# B&R Automation Studio project Panasonic_LinkaPowerCP2_A2021055 (part 31)

#### COM_Tester.st
```iecst
ACTION COM_Tester:

	//Parametre komunikácie//
    memcpy(ADR(SKTcpClientTester_0.Params.IPaddrServ),ADR('192.168.128.252'),SIZEOF('192.168.128.252'));
    (*memcpy(ADR(SKTcpClientTester_0.Params.IPaddrServ),ADR('127.0.0.1'),SIZEOF('127.0.0.1'));*)
    SKTcpClientTester_0.Params.IPportClient := P4_FunkcnyTestA.PAR.CisloPortuKlienta;
    SKTcpClientTester_0.Params.IPportServ := 1030;
    SKTcpClientTester_0.Params.RecvTimeout := 10000;
    strcpy(ADR(SKTcpClientTester_0.Params.Packet.data),ADR(dataStr));
    SKTcpClientTester_0();

    Cas_FunkcnyTestA.PT:= T#1M;
    Cas_FunkcnyTestA();

    //Volanie funkcie SequenceControl//
    SequenceControl(SC:= SC_OvlTesteraFT);

    CASE SC_OvlTesteraFT.Step OF

        0:
            SC_OvlTesteraFT.StepName:= '0 - Nulovanie';
            SKTcpClientTester_0.Enable:= TRUE;
            SKTcpClientTester_0.Cmd.Send:= FALSE;
			P4_FunkcnyTestA.STAV.TestovanieUkoncene:= FALSE;
			P4_FunkcnyTestA.STAV.TesterNeodpoveda:= FALSE;
            PocetDopytovNaTester:= 0;
            SC_OvlTesteraFT.ResetStep:= TRUE;
            SC_OvlTesteraFT.Step:= 1;

        1:
            SC_OvlTesteraFT.StepName:= '1 - Cakam na spustenie testera';
            IF P4_FunkcnyTestA.CMD.StartTestovania THEN
                P4_FunkcnyTestA.STAV.Vysledok_FV_Testu:= '';
                Cas_FunkcnyTestA.IN:= TRUE;
                NameranyCasFunkcnehoTestuA:= 0;
                SC_OvlTesteraFT.Step:= 10;
            END_IF

        10:
            SC_OvlTesteraFT.StepName:= '10 - Dopyt na stav testera - typ 0';
            SC_OvlTesteraFT.IdleTime.PT:= T#300ms;
            SC_OvlTesteraFT.AlarmTime.PT:= T#5s;
            SC_OvlTesteraFT.IdleTime.IN:= TRUE;
            SC_OvlTesteraFT.AlarmTime.IN:= TRUE;

            SKTcpClientTester_0.Params.Packet.type:= 0;
            SKTcpClientTester_0.Params.Packet.workplace:= 49;
            SKTcpClientTester_0.Params.Packet.id:= 1;
            SKTcpClientTester_0.Cmd.Close:= FALSE;
			SKTcpClientTester_0.Cmd.Send:= TRUE;

            IF SKTcpClientTester_0.Cmd.Send AND NOT SKTcpClientTester_0.Status.staReceived AND NOT SKTcpClientTester_0.Status.staError THEN
                SC_OvlTesteraFT.ResetStep:= TRUE;
                SC_OvlTesteraFT.Step:= 13;
            ELSIF SC_OvlTesteraFT.AlarmTime.Q AND (SKTcpClientTester_0.Status.staReceived OR SKTcpClientTester_0.Status.staError) THEN
                PocetDopytovNaTester:= PocetDopytovNaTester + 1;
				SKTcpClientTester_0.Cmd.Send:= FALSE;
				SKTcpClientTester_0.Cmd.Close:= TRUE;
				SC_OvlTesteraFT.ResetStep:= TRUE;
                SC_OvlTesteraFT.Step:= 12;
            END_IF

        12:
            SC_OvlTesteraFT.StepName:= '12 - Dopyt na stav testera - cakam na opatovny dopyt na tester';
            SC_OvlTesteraFT.IdleTime.PT:= T#800ms;
            SC_OvlTesteraFT.AlarmTime.PT:= T#5s;
            SC_OvlTesteraFT.IdleTime.IN:= TRUE;
            SKTcpClientTester_0.Cmd.Send:= FALSE;

            IF PocetDopytovNaTester < 10 THEN
                IF SC_OvlTesteraFT.IdleTime.Q THEN
                    SC_OvlTesteraFT.ResetStep:= TRUE;
                    SC_OvlTesteraFT.Step:= 10;
                END_IF
            ELSE
                P4_FunkcnyTestA.STAV.Vysledok_FV_Testu:= 'NG';
                P4_FunkcnyTestA.STAV.TesterNeodpoveda:= TRUE;
                SC_OvlTesteraFT.ResetStep:= TRUE;
                SC_OvlTesteraFT.Step:= 100;
            END_IF

        13:
            SC_OvlTesteraFT.StepName:= '13 - Odpoved na stav testera - typ 0';
            SC_OvlTesteraFT.IdleTime.PT:= T#800ms;
            SC_OvlTesteraFT.AlarmTime.PT:= T#10s;
            SC_OvlTesteraFT.IdleTime.IN:= TRUE;

            IF SKTcpClientTester_0.Status.staReceived AND SKTcpClientTester_0.Status.DataRecv[2]= 0 AND SKTcpClientTester_0.Status.DataRecv[5]= 2 THEN
                SKTcpClientTester_0.Cmd.Send:= FALSE;
                SC_OvlTesteraFT.ResetStep:= TRUE;
                SC_OvlTesteraFT.Step:= 15;
            ELSIF SKTcpClientTester_0.Status.staReceived AND SKTcpClientTester_0.Status.DataRecv[2]= 0 AND SKTcpClientTester_0.Status.DataRecv[5]= 1 THEN
				SKTcpClientTester_0.Cmd.Send:= FALSE;
				SKTcpClientTester_0.Cmd.Close:= TRUE;
                IF SC_OvlTesteraFT.IdleTime.Q THEN
                    SC_OvlTesteraFT.ResetStep:= TRUE;
                    SC_OvlTesteraFT.Step:= 10;
                END_IF
            ELSIF SKTcpClientTester_0.Status.staReceived AND SKTcpClientTester_0.Status.DataRecv[2]= 0 AND SKTcpClientTester_0.Status.DataRecv[5]= 0 THEN
                SKTcpClientTester_0.Cmd.Send:= FALSE;
                SKTcpClientTester_0.Cmd.Close:= TRUE;
				IF SC_OvlTesteraFT.IdleTime.Q THEN
                    SC_OvlTesteraFT.ResetStep:= TRUE;
                    SC_OvlTesteraFT.Step:= 10;
                END_IF
            ELSIF SKTcpClientTester_0.Status.staError THEN
                SKTcpClientTester_0.Cmd.Send:= FALSE;
                P4_FunkcnyTestA.STAV.Vysledok_FV_Testu:= 'NG';
                P4_FunkcnyTestA.STAV.TesterNeodpoveda:= TRUE;
                SC_OvlTesteraFT.ResetStep:= TRUE;
                SC_OvlTesteraFT.Step:= 100;
            END_IF

        15:
            SC_OvlTesteraFT.StepName:= '15 - Poslanie QR kodu Power CP - typ 1';
            SC_OvlTesteraFT.IdleTime.PT:= T#300ms;
            SC_OvlTesteraFT.AlarmTime.PT:= T#10s;
            SC_OvlTesteraFT.IdleTime.IN:= TRUE;

            SKTcpClientTester_0.Params.Packet.type:= 1;
            SKTcpClientTester_0.Params.Packet.workplace:= 49;
            SKTcpClientTester_0.Params.Packet.id:= 1;
			dataStr:= Paletka[i].PAR.QRkodPowerCP;
		    SKTcpClientTester_0.Cmd.Send:= TRUE;

            IF SKTcpClientTester_0.Cmd.Send AND NOT SKTcpClientTester_0.Status.staReceived AND NOT SKTcpClientTester_0.Status.staError THEN
                SC_OvlTesteraFT.ResetStep:= TRUE;
                SC_OvlTesteraFT.Step:= 18;
            END_IF

        18:
            SC_OvlTesteraFT.StepName:= '18 - Odpoved na poslanie QR kodu - typ 1';
            SC_OvlTesteraFT.IdleTime.PT:= T#300ms;
            SC_OvlTesteraFT.AlarmTime.PT:= T#10s;
            SC_OvlTesteraFT.IdleTime.IN:= TRUE;

            IF SKTcpClientTester_0.Status.staReceived AND SKTcpClientTester_0.Status.DataRecv[2]= 1 AND SKTcpClientTester_0.Status.DataRecv[5]= 0 THEN
                SKTcpClientTester_0.Cmd.Send:= FALSE;
                SC_OvlTesteraFT.ResetStep:= TRUE;
                SC_OvlTesteraFT.Step:= 20;
            ELSIF SKTcpClientTester_0.Status.staReceived AND SKTcpClientTester_0.Status.DataRecv[2]= 1 AND SKTcpClientTester_0.Status.DataRecv[5]= 2 THEN
                SKTcpClientTester_0.Cmd.Send:= FALSE;
                IF SC_OvlTesteraFT.IdleTime.Q THEN
                    SC_OvlTesteraFT.ResetStep:= TRUE;
                    SC_OvlTesteraFT.Step:= 15;
                END_IF
            ELSIF SKTcpClientTester_0.Status.staReceived AND SKTcpClientTester_0.Status.DataRecv[2]= 1 AND SKTcpClientTester_0.Status.DataRecv[5]= 1 THEN
                SKTcpClientTester_0.Cmd.Send:= FALSE;
                P4_FunkcnyTestA.STAV.Vysledok_FV_Testu:= 'NG';
                P4_FunkcnyTestA.STAV.TestovanieUkoncene:= TRUE;
                SC_OvlTesteraFT.ResetStep:= TRUE;
                SC_OvlTesteraFT.Step:= 100;
            ELSIF SKTcpClientTester_0.Status.staError THEN
                SKTcpClientTester_0.Cmd.Send:= FALSE;
                P4_FunkcnyTestA.STAV.Vysledok_FV_Testu:= 'NG';
                P4_FunkcnyTestA.STAV.TesterNeodpoveda:= TRUE;
                SC_OvlTesteraFT.ResetStep:= TRUE;
                SC_OvlTesteraFT.Step:= 100;
            END_IF

        20:
            SC_OvlTesteraFT.StepName:= '20 - Dopyt na stav testera - typ 0';
            SC_OvlTesteraFT.IdleTime.PT:= T#300ms;
            SC_OvlTesteraFT.AlarmTime.PT:= T#10s;
            SC_OvlTesteraFT.IdleTime.IN:= TRUE;

            SKTcpClientTester_0.Params.Packet.type:= 0;
            SKTcpClientTester_0.Params.Packet.workplace:= 49;
            SKTcpClientTester_0.Params.Packet.id:= 1;
            SKTcpClientTester_0.Cmd.Send:= TRUE;

            IF SKTcpClientTester_0.Cmd.Send AND NOT SKTcpClientTester_0.Status.staReceived AND NOT SKTcpClientTester_0.Status.staError THEN
                SC_OvlTesteraFT.ResetStep:= TRUE;
                SC_OvlTesteraFT.Step:= 23;
            END_IF

        23:
            SC_OvlTesteraFT.StepName:= '23 - Odpoved na stav testera - typ 0';
            SC_OvlTesteraFT.IdleTime.PT:= T#300ms;
            SC_OvlTesteraFT.AlarmTime.PT:= T#10s;
            SC_OvlTesteraFT.IdleTime.IN:= TRUE;

            IF SKTcpClientTester_0.Status.staReceived AND SKTcpClientTester_0.Status.DataRecv[2]= 0 AND SKTcpClientTester_0.Status.DataRecv[5]= 3 THEN
                SKTcpClientTester_0.Cmd.Send:= FALSE;
                IF SC_OvlTesteraFT.IdleTime.Q THEN
                    SC_OvlTesteraFT.ResetStep:= TRUE;
                    SC_OvlTesteraFT.Step:= 20;
                END_IF
            ELSIF SKTcpClientTester_0.Status.staReceived AND SKTcpClientTester_0.Status.DataRecv[2]= 0 AND SKTcpClientTester_0.Status.DataRecv[5]= 4 THEN
                SKTcpClientTester_0.Cmd.Send:= FALSE;
                SC_OvlTesteraFT.ResetStep:= TRUE;
                SC_OvlTesteraFT.Step:= 25;
            ELSIF SKTcpClientTester_0.Status.staReceived AND SKTcpClientTester_0.Status.DataRecv[2]= 0 AND SKTcpClientTester_0.Status.DataRecv[5]= 0 THEN
                SKTcpClientTester_0.Cmd.Send:= FALSE;
                P4_FunkcnyTestA.STAV.Vysledok_FV_Testu:= 'NG';
                P4_FunkcnyTestA.STAV.TestovanieUkoncene:= TRUE;
                SC_OvlTesteraFT.ResetStep:= TRUE;
                SC_OvlTesteraFT.Step:= 100;
            ELSIF SKTcpClientTester_0.Status.staError THEN
                SKTcpClientTester_0.Cmd.Send:= FALSE;
                P4_FunkcnyTestA.STAV.Vysledok_FV_Testu:= 'NG';
                P4_FunkcnyTestA.STAV.TesterNeodpoveda:= TRUE;
                SC_OvlTesteraFT.ResetStep:= TRUE;
                SC_OvlTesteraFT.Step:= 100;
            END_IF

        25:
            SC_OvlTesteraFT.StepName:= '25 - Dopyt na vysledok testu - typ 2';
            SC_OvlTesteraFT.IdleTime.PT:= T#300ms;
            SC_OvlTesteraFT.AlarmTime.PT:= T#10s;
            SC_OvlTesteraFT.IdleTime.IN:= TRUE;

            SKTcpClientTester_0.Params.Packet.type:= 2;
            SKTcpClientTester_0.Params.Packet.workplace:= 49;
            SKTcpClientTester_0.Params.Packet.id:= 1;
            SKTcpClientTester_0.Cmd.Send:= TRUE;

            IF SKTcpClientTester_0.Cmd.Send AND NOT SKTcpClientTester_0.Status.staReceived AND NOT SKTcpClientTester_0.Status.staError THEN
                SC_OvlTesteraFT.ResetStep:= TRUE;
                SC_OvlTesteraFT.Step:= 28;
            END_IF

        28:
            SC_OvlTesteraFT.StepName:= '28 - Odpoved na vysledok testu - typ 2';
            SC_OvlTesteraFT.IdleTime.PT:= T#300ms;
            SC_OvlTesteraFT.AlarmTime.PT:= T#10s;
            SC_OvlTesteraFT.IdleTime.IN:= TRUE;

            IF SKTcpClientTester_0.Status.staReceived AND SKTcpClientTester_0.Status.DataRecv[2]= 2 AND SKTcpClientTester_0.Status.DataRecv[5]= 1 THEN
                SKTcpClientTester_0.Cmd.Send:= FALSE;
                P4_FunkcnyTestA.STAV.Vysledok_FV_Testu:= 'OK';
                SC_OvlTesteraFT.ResetStep:= TRUE;
                SC_OvlTesteraFT.Step:= 30;
            ELSIF SKTcpClientTester_0.Status.staReceived AND SKTcpClientTester_0.Status.DataRecv[2]= 2 AND SKTcpClientTester_0.Status.DataRecv[5]= 2 THEN
                SKTcpClientTester_0.Cmd.Send:= FALSE;
                P4_FunkcnyTestA.STAV.Vysledok_FV_Testu:= 'NG';
                SC_OvlTesteraFT.ResetStep:= TRUE;
                SC_OvlTesteraFT.Step:= 30;
            ELSIF SKTcpClientTester_0.Status.staReceived AND SKTcpClientTester_0.Status.DataRecv[2]= 2 AND SKTcpClientTester_0.Status.DataRecv[5]= 0 THEN
                SKTcpClientTester_0.Cmd.Send:= FALSE;
                IF SC_OvlTesteraFT.IdleTime.Q THEN
                    SC_OvlTesteraFT.ResetStep:= TRUE;
                    SC_OvlTesteraFT.Step:= 25;
                END_IF
            ELSIF SKTcpClientTester_0.Status.staReceived AND SKTcpClientTester_0.Status.DataRecv[2]= 2 AND SKTcpClientTester_0.Status.DataRecv[5]= 3 THEN
                SKTcpClientTester_0.Cmd.Send:= FALSE;
                IF SC_OvlTesteraFT.IdleTime.Q THEN
                    SC_OvlTesteraFT.ResetStep:= TRUE;
                    SC_OvlTesteraFT.Step:= 25;
                END_IF
            ELSIF SKTcpClientTester_0.Status.staError THEN
                SKTcpClientTester_0.Cmd.Send:= FALSE;
                P4_FunkcnyTestA.STAV.Vysledok_FV_Testu:= 'NG';
                P4_FunkcnyTestA.STAV.TesterNeodpoveda:= TRUE;
                SC_OvlTesteraFT.ResetStep:= TRUE;
                SC_OvlTesteraFT.Step:= 100;
            END_IF

        30:
            SC_OvlTesteraFT.StepName:= '30 - Potvrdenie precitanie vysledkov testu - typ 3';
            SC_OvlTesteraFT.IdleTime.PT:= T#300ms;
            SC_OvlTesteraFT.AlarmTime.PT:= T#10s;
            SC_OvlTesteraFT.IdleTime.IN:= TRUE;

            SKTcpClientTester_0.Params.Packet.type:= 3;
            SKTcpClientTester_0.Params.Packet.workplace:= 49;
            SKTcpClientTester_0.Params.Packet.id:= 1;
            SKTcpClientTester_0.Cmd.Send:= TRUE;

            IF SKTcpClientTester_0.Cmd.Send AND NOT SKTcpClientTester_0.Status.staReceived AND NOT SKTcpClientTester_0.Status.staError THEN
                SC_OvlTesteraFT.ResetStep:= TRUE;
                SC_OvlTesteraFT.Step:= 33;
            END_IF

        33:
            SC_OvlTesteraFT.StepName:= '33 - Odpoved testera na potvrdenie vysledkov - typ 3';
            SC_OvlTesteraFT.IdleTime.PT:= T#500ms;
            SC_OvlTesteraFT.AlarmTime.PT:= T#10s;

            IF SKTcpClientTester_0.Status.staReceived AND SKTcpClientTester_0.Status.DataRecv[2]= 3 AND SKTcpClientTester_0.Status.DataRecv[5]= 0 THEN
                SKTcpClientTester_0.Cmd.Send:= FALSE;
                P4_FunkcnyTestA.STAV.TestovanieUkoncene:= TRUE;
                SC_OvlTesteraFT.ResetStep:= TRUE;
                SC_OvlTesteraFT.Step:= 100;
            ELSIF SKTcpClientTester_0.Status.staReceived AND SKTcpClientTester_0.Status.DataRecv[2]= 3 AND SKTcpClientTester_0.Status.DataRecv[5]= 1 THEN
                P4_FunkcnyTestA.STAV.Vysledok_FV_Testu:= 'NG';
                P4_FunkcnyTestA.STAV.TestovanieUkoncene:= TRUE;
                SKTcpClientTester_0.Cmd.Send:= FALSE;
                SC_OvlTesteraFT.ResetStep:= TRUE;
                SC_OvlTesteraFT.Step:= 100;
            ELSIF SKTcpClientTester_0.Status.staError THEN
                SKTcpClientTester_0.Cmd.Send:= FALSE;
				P4_FunkcnyTestA.STAV.Vysledok_FV_Testu:= 'NG';
				P4_FunkcnyTestA.STAV.TesterNeodpoveda:= TRUE;
				SC_OvlTesteraFT.ResetStep:= TRUE;
                SC_OvlTesteraFT.Step:= 100;
            END_IF

        100:
            SC_OvlTesteraFT.StepName:= '100 - Cakam na zrusenie signalu start testovania';
            SC_OvlTesteraFT.IdleTime.PT:= T#3s;
            SC_OvlTesteraFT.AlarmTime.PT:= T#10s;

            NameranyCasFunkcnehoTestuA:= Cas_FunkcnyTestA.ET;
            Cas_FunkcnyTestA.IN:= FALSE;

            IF NOT P4_FunkcnyTestA.CMD.StartTestovania THEN
                SC_OvlTesteraFT.ResetStep:= TRUE;
                SC_OvlTesteraFT.Step:= 0;
            END_IF

    END_CASE

END_ACTION
```

### Program Logical/Program/Pracovisko_4/P4_FunkcnyTestB (IEC)

#### Main.st - Init, cyclic, exit code
```iecst
PROGRAM _INIT
	P4_FunkcnyTestB.PAR.CisloPortuKlienta:= 1050;

END_PROGRAM

PROGRAM _CYCLIC

	//Volanie funkcie SequenceControl//
	SequenceControl(SC:= SC_P4_FunkcnyTestB);

	//Volanie podprogramov//
	OvlCentrovacky;
	OvlHornychKontaktov;
	OvlSpodnychKontaktov;
	IOLinkKomunikacia;
	COM_Tester;

	//Reset sekcie //
	IF P4_FunkcnyTestB.Reset THEN
		SC_P4_FunkcnyTestB.Step:= 0;
		P4_FunkcnyTestB.Reset:= FALSE;
	ELSIF NOT Safety.STAV.Linka_ZonaCS_AKTIVNA THEN
		SC_P4_FunkcnyTestB.Step:= 0;
	END_IF

	CASE SC_P4_FunkcnyTestB.Step OF

		0:
			SC_P4_FunkcnyTestB.StepName:='0 - Nulovanie';
			SC_OvlCentrovacky.Step:= 0;
			SC_OvlHornychKontaktov.Step:= 0;
			SC_OvlSpodnychKontaktov.Step:= 0;
			SC_OvlTesteraFT.Step:= 0;
			P4_FunkcnyTestB.Automat:= FALSE;
			P4_FunkcnyTestB.KoniecCyklu:= FALSE;
			P4_FunkcnyTestB.Manual:= FALSE;
			P4_FunkcnyTestB.STAV.PoINIT:= FALSE;
			P4_FunkcnyTestB.OUT.ZasunStoper:= FALSE;
			P4_FunkcnyTestB.OUT.KontaktyTestera_VYSUN:= FALSE;
			P4_FunkcnyTestB.OUT.OdpruzHornychKontaktov_VYSUN:= FALSE;
			P4_FunkcnyTestB.OUT.OdpruzHornychKontaktov_ZASUN:= TRUE;
			P4_FunkcnyTestB.OUT.PritlakPowerCP_VYSUN:= FALSE;
			P4_FunkcnyTestB.OUT.SpodneKontakty_VYSUN:= FALSE;
			P4_FunkcnyTestB.OUT.SpodneKontakty_ZASUN:= TRUE;
			P4_FunkcnyTestB.OUT.HorneKontakty_VYSUN:= FALSE;
			P4_FunkcnyTestB.OUT.HorneKontakty_ZASUN:= TRUE;
			P4_FunkcnyTestB.RFID_hlava.PrecitajChipRFID:= FALSE;
			P4_FunkcnyTestB.CMD.RR_ZatvorTester:= FALSE;
			P4_FunkcnyTestB.CMD.StartTestovania:= FALSE;
			P4_FunkcnyTestB.CMD.RR_VysunPruzenieKontaktov:= FALSE;
			P4_FunkcnyTestB.CMD.OpatovnyTest:= FALSE;
			P4_FunkcnyTestB.STAV.RR_SekvenciaTestera_BUSY:= FALSE;
			P4_FunkcnyTestB.STAV.PaletkaOznacena_NG:= FALSE;
			P34_Vizu.ZobrazHL1_FinalTestB:= FALSE;
			P3_ZdvizkaZaLeakTestB.STAV.PrebiehaVyvezeniePaletkyNaTratB:= FALSE;
			P4_FunkcnyTestB.STAV.PrebiehaVyvezeniePaletky:= FALSE;
			TestovaciKus:= FALSE;
			P4_FinalTestB_Taktime.IN.START_MeraniaCasu:= FALSE;
			P4_FinalTestB_Taktime.IN.START_MeraniaStratovehoCasu:= FALSE;

			PocetDopytovNaTester:= 0;

			IF Safety.STAV.Linka_ZonaCS_AKTIVNA AND
				Safety.STAV.P4_ZonaBunky_AKTIVNA AND
				P4_Pracovisko.STAV.HardwareBunky_OK AND
				NOT P4_Pracovisko.STAV.Porucha_ST1 AND
				NOT P4_Pracovisko.STAV.Porucha_ST2 AND
				NOT P4_Pracovisko.STAV.Porucha_ST3 AND
				NOT P4_Pracovisko.STAV.Porucha_ST4 AND
				NOT P4_Pracovisko.STAV.Porucha_ST5 AND
				NOT P4_Pracovisko.STAV.Porucha_ST6 THEN
				SC_P4_FunkcnyTestB.ResetStep:= TRUE;
				SC_P4_FunkcnyTestB.Step:= 1;
			END_IF

		1:
			SC_P4_FunkcnyTestB.StepName:='1 - Cakam na spustenie vyroby';
			P4_FunkcnyTestB.KoniecCyklu:= FALSE;
			IF P4_FunkcnyTestB.Automat THEN
				SC_P4_FunkcnyTestB.Step:= 2;
			ELSIF P4_FunkcnyTestB.Manual THEN
				SC_P4_FunkcnyTestB.Step:= 700;
			END_IF

			//********************************************************Inicializácia****************************************************************************//

		2:
			SC_P4_FunkcnyTestB.StepName:='2 - Inicializacia - cakam na spustenie inicializacie';
			SC_P4_FunkcnyTestB.IdleTime.PT:= T#500ms;
			SC_P4_FunkcnyTestB.AlarmTime.PT:= T#5s;

			SC_P4_FunkcnyTestB.IdleTime.IN:= TRUE;

			IF SC_P4_FunkcnyTestB.IdleTime.Q THEN
				SC_P4_FunkcnyTestB.ResetStep:= TRUE;
				SC_P4_FunkcnyTestB.Step:= 5;
			END_IF

		5:
			SC_P4_FunkcnyTestB.StepName:='5 - Inicializacia - zasunutie spodnych kontaktov';
			SC_P4_FunkcnyTestB.IdleTime.PT:= T#4s;
			SC_P4_FunkcnyTestB.AlarmTime.PT:= T#5s;

			IF NOT SC_P4_FunkcnyTestB.Switch1 THEN
				SpodneKontakty_ZASUN:= TRUE;
				SC_P4_FunkcnyTestB.Switch1:= TRUE;
			END_IF

			IF P4_FunkcnyTestB.IN.SpodneKontakty_ZASUNUTE THEN
				SC_P4_FunkcnyTestB.ResetStep:= TRUE;
				SC_P4_FunkcnyTestB.Step:= 8;
			END_IF

		8:
			SC_P4_FunkcnyTestB.StepName:='8 - Inicializacia - zasunutie hornych kontaktov';
			SC_P4_FunkcnyTestB.IdleTime.PT:= T#4s;
			SC_P4_FunkcnyTestB.AlarmTime.PT:= T#5s;

			IF NOT SC_P4_FunkcnyTestB.Switch1 THEN
				HorneKontakty_ZASUN:= TRUE;
				SC_P4_FunkcnyTestB.Switch1:= TRUE;
			END_IF

			IF P4_FunkcnyTestB.IN.HorneKontakty_ZASUNUTE THEN
				SC_P4_FunkcnyTestB.ResetStep:= TRUE;
				SC_P4_FunkcnyTestB.Step:= 10;
			END_IF

		10:
			SC_P4_FunkcnyTestB.StepName:='10 - Inicializacia - zasunutie cenrovacky';
			SC_P4_FunkcnyTestB.IdleTime.PT:= T#4s;
			SC_P4_FunkcnyTestB.AlarmTime.PT:= T#5s;

			IF NOT SC_P4_FunkcnyTestB.Switch1 THEN
				Centrovacku_ZASUN:= TRUE;
				SC_P4_FunkcnyTestB.Switch1:= TRUE;
			END_IF

			IF P4_FunkcnyTestB.IN.Centrovanie_ZASUNUTE THEN
				SC_P4_FunkcnyTestB.ResetStep:= TRUE;
				SC_P4_FunkcnyTestB.Step:= 13;
			END_IF

		13:
			SC_P4_FunkcnyTestB.StepName:='13 - Inicializacia - kontrola kontaktov Funkcneho testu';
			SC_P4_FunkcnyTestB.IdleTime.PT:= T#4s;
			SC_P4_FunkcnyTestB.AlarmTime.PT:= T#5s;

			IF Linka.PAR.ZvolenyModel = '4F' AND P4_FunkcnyTestB.IN.TypSpodnychKontaktov_4F THEN
				SC_P4_FunkcnyTestB.ResetStep:= TRUE;
				SC_P4_FunkcnyTestB.Step:= 15;
			ELSIF Linka.PAR.ZvolenyModel = '5F' AND P4_FunkcnyTestB.IN.TypSpodnychKontaktov_5F_5H THEN
				SC_P4_FunkcnyTestB.ResetStep:= TRUE;
				SC_P4_FunkcnyTestB.Step:= 15;
			ELSIF Linka.PAR.ZvolenyModel = '5H' AND P4_FunkcnyTestB.IN.TypSpodnychKontaktov_5F_5H THEN
				SC_P4_FunkcnyTestB.ResetStep:= TRUE;
				SC_P4_FunkcnyTestB.Step:= 15;
			ELSE
				P34_Alarmy[438]:= TRUE;
				P4_Pracovisko.STAV.Porucha_ST2:= TRUE;
			END_IF

		15:
			SC_P4_FunkcnyTestB.StepName:='15 - Inicializacia - hladanie paletky';
			SC_P4_FunkcnyTestB.IdleTime.PT:= T#5s;
			SC_P4_FunkcnyTestB.AlarmTime.PT:= T#5s;

			SC_P4_FunkcnyTestB.IdleTime.IN:= P4_Dopravniky.STAV.PoINIT;

			IF P4_FunkcnyTestB.RFID_hlava.PritomnostPaletky THEN
				SC_P4_FunkcnyTestB.ResetStep:= TRUE;
				SC_P4_FunkcnyTestB.Step:= 20;
			ELSIF SC_P4_FunkcnyTestB.IdleTime.Q THEN
				P4_FunkcnyTestB.STAV.PoINIT:= TRUE;
				SC_P4_FunkcnyTestB.ResetStep:= TRUE;
				SC_P4_FunkcnyTestB.Step:= 100;
			END_IF

		20:
			SC_P4_FunkcnyTestB.StepName:='20 - Inicializacia - precitanie cisla paletky';
			SC_P4_FunkcnyTestB.IdleTime.PT:= T#200ms;
			SC_P4_FunkcnyTestB.AlarmTime.PT:= T#5s;

			SC_P4_FunkcnyTestB.IdleTime.IN:= P4_FunkcnyTestB.RFID_hlava.PritomnostPaletky;

			IF SC_P4_FunkcnyTestB.IdleTime.Q AND NOT SC_P4_FunkcnyTestB.Switch1 THEN
				P4_FunkcnyTestB.RFID_hlava.PrecitajChipRFID:= TRUE;
				i:= 0;
				SC_P4_FunkcnyTestB.Switch1:= TRUE;
			END_IF

			IF P4_FunkcnyTestB.RFID_hlava.Stav_CitanieZapis_OK AND P4_FunkcnyTestB.RFID_hlava.PrecitaneCisloPaletky <> 0 THEN
				i:= P4_FunkcnyTestB.RFID_hlava.PrecitaneCisloPaletky;
				P4_FunkcnyTestB.RFID_hlava.PrecitajChipRFID:= FALSE;
				SC_P4_FunkcnyTestB.ResetStep:= TRUE;
				SC_P4_FunkcnyTestB.Step:= 23;
			END_IF

		23:
			SC_P4_FunkcnyTestB.StepName:='23 - Inicializacia - priradenie indexu paletky na zaklade precitanej hodnoty';
			SC_P4_FunkcnyTestB.IdleTime.PT:= T#200ms;
			SC_P4_FunkcnyTestB.AlarmTime.PT:= T#5s;

			IF i<> 0 THEN
				P4_FunkcnyTestB.PAR.CisloPaletky_STRING:= USINT_TO_STRING(i);
				Paletka[i].PAR.CisloPaletky:= USINT_TO_STRING(i);
				SC_P4_FunkcnyTestB.ResetStep:= TRUE;
				SC_P4_FunkcnyTestB.Step:= 30;
			ELSE
				P34_Alarmy[429]:= TRUE;
				P4_Pracovisko.STAV.Porucha_ST2:= TRUE;
			END_IF

		30:
			SC_P4_FunkcnyTestB.StepName:='30 - Inicializacia - kontrola stavu paletky';
			SC_P4_FunkcnyTestB.IdleTime.PT:= T#200ms;
			SC_P4_FunkcnyTestB.AlarmTime.PT:= T#5s;

			IF Paletka[i].STAV.StavPaletky = '' THEN
				Paletka[i].STAV.StavPaletky:= 'NG';
				SC_P4_FunkcnyTestB.ResetStep:= TRUE;
				SC_P4_FunkcnyTestB.Step:= 560;
			ELSIF Paletka[i].STAV.StavPaletky = 'PRECH' THEN
				P4_FunkcnyTestB.STAV.PoINIT:= TRUE;
				SC_P4_FunkcnyTestB.ResetStep:= TRUE;
				SC_P4_FunkcnyTestB.Step:= 560;
			ELSIF Paletka[i].STAV.StavPaletky = 'TEST' AND Paletka[i].STAV.CisloTestovacejStanice = 'ST_FT1,FT2' THEN
				TestovaciKus:= TRUE;
				P4_FunkcnyTestB.STAV.PoINIT:= TRUE;
				SC_P4_FunkcnyTestB.ResetStep:= TRUE;
				SC_P4_FunkcnyTestB.Step:= 110;
			ELSIF Paletka[i].STAV.StavPaletky = 'TEST' AND Paletka[i].STAV.CisloTestovacejStanice <> 'ST_FT1,FT2' THEN
				P4_FunkcnyTestB.STAV.PoINIT:= TRUE;
				SC_P4_FunkcnyTestB.ResetStep:= TRUE;
				SC_P4_FunkcnyTestB.Step:= 560;
			ELSIF Paletka[i].STAV.StavPaletky = 'REV' AND Paletka[i].STAV.CisloRevorkovejStanice = 'ST_FT1,FT2' THEN
				IF P4_FunkcnyTestB.STAV.Tester_ON THEN
					Paletka[i].STAV.StavPaletky:= 'OK';
					P4_FunkcnyTestB.STAV.PoINIT:= TRUE;
					SC_P4_FunkcnyTestB.ResetStep:= TRUE;
					SC_P4_FunkcnyTestB.Step:= 110;
				ELSE
					P4_FunkcnyTestB.STAV.PoINIT:= TRUE;
					SC_P4_FunkcnyTestB.ResetStep:= TRUE;
					SC_P4_FunkcnyTestB.Step:= 560;
				END_IF
			ELSIF Paletka[i].STAV.StavPaletky = 'REV' AND Paletka[i].STAV.CisloRevorkovejStanice <> 'ST_FT1,FT2' THEN
				P4_FunkcnyTestB.STAV.PoINIT:= TRUE;
				SC_P4_FunkcnyTestB.ResetStep:= TRUE;
				SC_P4_FunkcnyTestB.Step:= 560;
			ELSIF Paletka[i].STAV.StavPaletky = 'OK' THEN
				SC_P4_FunkcnyTestB.ResetStep:= TRUE;
				SC_P4_FunkcnyTestB.Step:= 33;
			ELSIF Paletka[i].STAV.StavPaletky = 'NG' THEN
				P4_FunkcnyTestB.STAV.PoINIT:= TRUE;
				SC_P4_FunkcnyTestB.ResetStep:= TRUE;
				SC_P4_FunkcnyTestB.Step:= 560;
			END_IF

		33:
			SC_P4_FunkcnyTestB.StepName:='33 - Inicializacia - kontrola ukonceneho HV testu';
			SC_P4_FunkcnyTestB.IdleTime.PT:= T#200ms;
			SC_P4_FunkcnyTestB.AlarmTime.PT:= T#5s;

			IF Paletka[i].STAV.FunkcnyTest_Ukonceny THEN
				P4_FunkcnyTestB.STAV.PoINIT:= TRUE;
				SC_P4_FunkcnyTestB.ResetStep:= TRUE;
				SC_P4_FunkcnyTestB.Step:= 560;
			ELSE
				P4_FunkcnyTestB.STAV.PoINIT:= TRUE;
				SC_P4_FunkcnyTestB.ResetStep:= TRUE;
				SC_P4_FunkcnyTestB.Step:= 110;
			END_IF

		//********************************************************Automatický režim****************************************************************************//

		100:
			SC_P4_FunkcnyTestB.StepName:='100 - Automaticky Rezim - cakam na príchod paletky na stoper';
			SC_P4_FunkcnyTestB.IdleTime.PT:= T#200ms;
			SC_P4_FunkcnyTestB.AlarmTime.PT:= T#5s;

			SC_P4_FunkcnyTestB.IdleTime.IN:= P4_FunkcnyTestB.RFID_hlava.PritomnostPaletky;

			IF P4_FunkcnyTestB.RFID_hlava.PritomnostPaletky THEN
				P3_ZdvizkaZaLeakTestB.STAV.PrebiehaVyvezeniePaletkyNaTratB:= FALSE;
			END_IF

			IF NOT SC_P4_FunkcnyTestB.Switch1 AND P4_FunkcnyTestB.RFID_hlava.PritomnostPaletky THEN
				P4_FinalTestB_Taktime.IN.START_MeraniaCasu:= TRUE;
				P4_FinalTestB_Taktime.IN.ZAPIS_MeraniaCasu:= TRUE;
				P4_FinalTestB_Taktime.IN.ZAPIS_StratovyCas:= TRUE;
				Buffer_12.Hodnota:= P4_FinalTestB_Taktime.OUT.StratoveSekundy;
				Buffer_12.ZapisHodnotu:= TRUE;
				SC_P4_FunkcnyTestB.Switch1:= TRUE;
			END_IF

			IF P4_FunkcnyTestB.KoniecCyklu THEN
				SC_P4_FunkcnyTestB.ResetStep:= TRUE;
				SC_P4_FunkcnyTestB.Step:= 0;
			ELSIF SC_P4_FunkcnyTestB.IdleTime.Q THEN
				SC_P4_FunkcnyTestB.ResetStep:= TRUE;
				SC_P4_FunkcnyTestB.Step:= 101;
			END_IF

		101:
			SC_P4_FunkcnyTestB.StepName:='101 - Automaticky Rezim - precitanie cisla paletky';
			SC_P4_FunkcnyTestB.IdleTime.PT:= T#200ms;
			SC_P4_FunkcnyTestB.AlarmTime.PT:= T#5s;
			SC_P4_FunkcnyTestB.IdleTime.IN:= TRUE;

			IF NOT SC_P4_FunkcnyTestB.Switch1 THEN
				P4_FunkcnyTestB.RFID_hlava.PrecitajChipRFID:= TRUE;
				i:= 0;
				SC_P4_FunkcnyTestB.Switch1:= TRUE;
			END_IF

			IF P4_FunkcnyTestB.RFID_hlava.Stav_CitanieZapis_OK AND P4_FunkcnyTestB.RFID_hlava.PrecitaneCisloPaletky <> 0 THEN
				i:= P4_FunkcnyTestB.RFID_hlava.PrecitaneCisloPaletky;
				P4_FunkcnyTestB.RFID_hlava.PrecitajChipRFID:= FALSE;
				SC_P4_FunkcnyTestB.ResetStep:= TRUE;
				SC_P4_FunkcnyTestB.Step:= 102;
			END_IF

		102:
			SC_P4_FunkcnyTestB.StepName:='102 - Automaticky Rezim - priradenie indexu paletky na zaklade precitanej hodnoty';
			SC_P4_FunkcnyTestB.IdleTime.PT:= T#200ms;
			SC_P4_FunkcnyTestB.AlarmTime.PT:= T#5s;

			IF i<> 0 THEN
				P4_FunkcnyTestB.PAR.CisloPaletky_STRING:= USINT_TO_STRING(i);
				Paletka[i].PAR.CisloPaletky:= USINT_TO_STRING(i);
				SC_P4_FunkcnyTestB.ResetStep:= TRUE;
				SC_P4_FunkcnyTestB.Step:= 103;
			ELSE
				P34_Alarmy[429]:= TRUE;
				P4_Pracovisko.STAV.Porucha_ST2:= TRUE;
			END_IF

		103:
			SC_P4_FunkcnyTestB.StepName:='103 - Automaticky Rezim - kontrola stavu paletky';
			SC_P4_FunkcnyTestB.IdleTime.PT:= T#200ms;
			SC_P4_FunkcnyTestB.AlarmTime.PT:= T#5s;

			IF Paletka[i].STAV.StavPaletky = '' THEN
				Paletka[i].STAV.StavPaletky:= 'NG';
				SC_P4_FunkcnyTestB.ResetStep:= TRUE;
				SC_P4_FunkcnyTestB.Step:= 560;
			ELSIF Paletka[i].STAV.StavPaletky = 'PRECH' THEN
				SC_P4_FunkcnyTestB.ResetStep:= TRUE;
				SC_P4_FunkcnyTestB.Step:= 560;
			ELSIF Paletka[i].STAV.StavPaletky = 'TEST' AND Paletka[i].STAV.CisloTestovacejStanice = 'ST_FT1,FT2' THEN
				TestovaciKus:= TRUE;
				SC_P4_FunkcnyTestB.ResetStep:= TRUE;
				SC_P4_FunkcnyTestB.Step:= 110;
			ELSIF Paletka[i].STAV.StavPaletky = 'TEST' AND Paletka[i].STAV.CisloTestovacejStanice <> 'ST_FT1,FT2' THEN
				SC_P4_FunkcnyTestB.ResetStep:= TRUE;
				SC_P4_FunkcnyTestB.Step:= 560;
			ELSIF Paletka[i].STAV.StavPaletky = 'REV' AND Paletka[i].STAV.CisloRevorkovejStanice = 'ST_FT1,FT2' THEN
				IF P4_FunkcnyTestB.STAV.Tester_ON THEN
					Paletka[i].STAV.StavPaletky:= 'OK';
					SC_P4_FunkcnyTestB.ResetStep:= TRUE;
					SC_P4_FunkcnyTestB.Step:= 110;
				ELSE
					SC_P4_FunkcnyTestB.ResetStep:= TRUE;
					SC_P4_FunkcnyTestB.Step:= 560;
				END_IF
			ELSIF Paletka[i].STAV.StavPaletky = 'REV' AND Paletka[i].STAV.CisloRevorkovejStanice <> 'ST_FT1,FT2' THEN
				SC_P4_FunkcnyTestB.ResetStep:= TRUE;
				SC_P4_FunkcnyTestB.Step:= 560;
			ELSIF Paletka[i].STAV.StavPaletky = 'OK' THEN
				SC_P4_FunkcnyTestB.ResetStep:= TRUE;
				SC_P4_FunkcnyTestB.Step:= 110;
			ELSIF Paletka[i].STAV.StavPaletky = 'NG' THEN
				SC_P4_FunkcnyTestB.ResetStep:= TRUE;
				SC_P4_FunkcnyTestB.Step:= 560;
			END_IF

		//Zatvorenie Funkčného testera//

		110:
			SC_P4_FunkcnyTestB.StepName:='110 - Automaticky Rezim - zacentrovanie paletky';
			SC_P4_FunkcnyTestB.IdleTime.PT:= T#200ms;
			SC_P4_FunkcnyTestB.AlarmTime.PT:= T#5s;

			IF NOT SC_P4_FunkcnyTestB.Switch1 THEN
				Centrovacku_VYSUN:= TRUE;
				SC_P4_FunkcnyTestB.Switch1:= TRUE;
			END_IF

			IF P4_FunkcnyTestB.IN.Centrovanie_VYSUNUTE THEN
				SC_P4_FunkcnyTestB.ResetStep:= TRUE;
				SC_P4_FunkcnyTestB.Step:= 113;
			END_IF

		113:
			SC_P4_FunkcnyTestB.StepName:='113 - Automaticky Rezim - vysunutie pruzenia hornych kontaktov';
			SC_P4_FunkcnyTestB.IdleTime.PT:= T#500ms;
			SC_P4_FunkcnyTestB.AlarmTime.PT:= T#5s;

			IF NOT SC_P4_FunkcnyTestB.Switch1 THEN
				P4_FunkcnyTestB.OUT.OdpruzHornychKontaktov_ZASUN:= FALSE;
				P4_FunkcnyTestB.OUT.OdpruzHornychKontaktov_VYSUN:= TRUE;
				SC_P4_FunkcnyTestB.IdleTime.IN:= TRUE;
				SC_P4_FunkcnyTestB.Switch1:= TRUE;
			END_IF

			IF SC_P4_FunkcnyTestB.IdleTime.Q THEN
				SC_P4_FunkcnyTestB.ResetStep:= TRUE;
				SC_P4_FunkcnyTestB.Step:= 115;
			END_IF

		115:
			SC_P4_FunkcnyTestB.StepName:='115 - Automaticky Rezim - vysunutie hornych kontaktov';
			SC_P4_FunkcnyTestB.IdleTime.PT:= T#200ms;
			SC_P4_FunkcnyTestB.AlarmTime.PT:= T#5s;

			IF NOT SC_P4_FunkcnyTestB.Switch1 THEN
				HorneKontakty_VYSUN:= TRUE;
				SC_P4_FunkcnyTestB.Switch1:= TRUE;
			END_IF

			IF P4_FunkcnyTestB.IN.HorneKontakty_VYSUNUTE THEN
				SC_P4_FunkcnyTestB.ResetStep:= TRUE;
				SC_P4_FunkcnyTestB.Step:= 118;
			END_IF

		118:
			SC_P4_FunkcnyTestB.StepName:='118 - Automaticky Rezim - vysunutie spodnych kontaktov';
			SC_P4_FunkcnyTestB.IdleTime.PT:= T#200ms;
			SC_P4_FunkcnyTestB.AlarmTime.PT:= T#5s;

			IF NOT SC_P4_FunkcnyTestB.Switch1 THEN
				SpodneKontakty_VYSUN:= TRUE;
				SC_P4_FunkcnyTestB.Switch1:= TRUE;
			END_IF

			IF P4_FunkcnyTestB.IN.SpodneKontakty_VYSUNUTE THEN
				SC_P4_FunkcnyTestB.ResetStep:= TRUE;
				SC_P4_FunkcnyTestB.Step:= 120;
			END_IF

		120:
			SC_P4_FunkcnyTestB.StepName:='120 - Automaticky Rezim - pritlacenie kontaktov testera';
			SC_P4_FunkcnyTestB.IdleTime.PT:= T#1s;
			SC_P4_FunkcnyTestB.AlarmTime.PT:= T#5s;

			P4_FunkcnyTestB.OUT.KontaktyTestera_VYSUN:= TRUE;
			SC_P4_FunkcnyTestB.IdleTime.IN:= TRUE;

			IF SC_P4_FunkcnyTestB.IdleTime.Q THEN
				IF P4_FunkcnyTestB.Manual THEN
					IF NOT P4_FunkcnyTestB.CMD.RR_ZatvorTester THEN
						SC_P4_FunkcnyTestB.ResetStep:= TRUE;
						SC_P4_FunkcnyTestB.Step:= 140;
					END_IF
				ELSE
					SC_P4_FunkcnyTestB.ResetStep:= TRUE;
					SC_P4_FunkcnyTestB.Step:= 130;
				END_IF
			END_IF

		130:
			SC_P4_FunkcnyTestB.StepName:='130 - Automaticky Rezim - spustenie testera';
			SC_P4_FunkcnyTestB.IdleTime.PT:= T#2s;
			SC_P4_FunkcnyTestB.AlarmTime.PT:= T#5s;

			SC_P4_FunkcnyTestB.IdleTime.IN:= TRUE;

			IF Linka.KOM_Panatrace_OFF THEN
				IF SC_P4_FunkcnyTestB.IdleTime.Q THEN
					SC_P4_FunkcnyTestB.ResetStep:= TRUE;
					SC_P4_FunkcnyTestB.Step:= 140;
				END_IF
			ELSE
				P4_FunkcnyTestB.STAV.Vysledok_FV_Testu:= '';
				P4_FunkcnyTestB.CMD.StartTestovania:= TRUE;
				P4_FinalTestB_Taktime.IN.START_MeraniaStratovehoCasu:= TRUE;
				SC_P4_FunkcnyTestB.ResetStep:= TRUE;
				SC_P4_FunkcnyTestB.Step:= 133;
			END_IF

		133:
			SC_P4_FunkcnyTestB.StepName:='133 - Automaticky Rezim - cakam na ukoncenie HV testu';
			SC_P4_FunkcnyTestB.IdleTime.PT:= T#1s;
			SC_P4_FunkcnyTestB.AlarmTime.PT:= T#5s;

			IF P4_FunkcnyTestB.STAV.TestovanieUkoncene THEN
				P4_FinalTestB_Taktime.IN.START_MeraniaStratovehoCasu:= FALSE;
				Paletka[i].STAV.FunkcnyTest_Ukonceny:= TRUE;
				P4_FunkcnyTestB.CMD.StartTestovania:= FALSE;
				IF Paletka[i].STAV.StavPaletky = 'TEST' THEN
					SC_P4_FunkcnyTestB.ResetStep:= TRUE;
					SC_P4_FunkcnyTestB.Step:= 135;
				ELSE
					IF P4_FunkcnyTestB.STAV.Vysledok_FV_Testu = 'OK' THEN
						Paletka[i].STAV.StavPaletky:= 'OK';
					ELSIF P4_FunkcnyTestB.STAV.Vysledok_FV_Testu = 'NG' THEN
						Paletka[i].STAV.StavPaletky:= 'NG';
					END_IF
					SC_P4_FunkcnyTestB.ResetStep:= TRUE;
					SC_P4_FunkcnyTestB.Step:= 135;
				END_IF
			ELSIF P4_FunkcnyTestB.STAV.TesterNeodpoveda THEN
				P4_FunkcnyTestB.CMD.StartTestovania:= FALSE;
				SC_P4_FunkcnyTestB.ResetStep:= TRUE;
				SC_P4_FunkcnyTestB.Step:= 134;
			END_IF

		134:
			SC_P4_FunkcnyTestB.StepName:='134 - Automaticky Rezim - zobrazenie hlasenia tester neodpoveda';
			SC_P4_FunkcnyTestB.IdleTime.PT:= T#1s;
			SC_P4_FunkcnyTestB.AlarmTime.PT:= T#5s;

			P34_Vizu.ZobrazHL1_FinalTestB:= TRUE;

			IF P4_FunkcnyTestB.CMD.OpatovnyTest THEN
				P4_FunkcnyTestB.CMD.OpatovnyTest:= FALSE;
				P34_Vizu.ZobrazHL1_FinalTestB:= FALSE;
				IF P4_FunkcnyTestB.PAR.CisloPortuKlienta < 1059 THEN
					P4_FunkcnyTestB.PAR.CisloPortuKlienta:= P4_FunkcnyTestB.PAR.CisloPortuKlienta + 1;
				ELSE
					P4_FunkcnyTestB.PAR.CisloPortuKlienta:= 1050;
				END_IF
				SC_P4_FunkcnyTestB.ResetStep:= TRUE;
				SC_P4_FunkcnyTestB.Step:= 130;
			ELSIF P4_FunkcnyTestB.STAV.PaletkaOznacena_NG THEN
				P4_FunkcnyTestB.STAV.PaletkaOznacena_NG:= FALSE;
				P34_Vizu.ZobrazHL1_FinalTestB:= FALSE;
				Paletka[i].STAV.StavPaletky:= 'NG';
				SC_P4_FunkcnyTestB.ResetStep:= TRUE;
				SC_P4_FunkcnyTestB.Step:= 135;
			END_IF

		135:
			SC_P4_FunkcnyTestB.StepName:='135 - Automaticky Rezim - cakam na zrusenie signalu Funkcny test ukonceny';
			SC_P4_FunkcnyTestB.IdleTime.PT:= T#1s;
			SC_P4_FunkcnyTestB.AlarmTime.PT:= T#5s;

			IF NOT P4_FunkcnyTestB.STAV.TestovanieUkoncene THEN
				SC_P4_FunkcnyTestB.ResetStep:= TRUE;
				SC_P4_FunkcnyTestB.Step:= 140;
			END_IF

		//Otvorenie Funkcneho testera//

		140:
			SC_P4_FunkcnyTestB.StepName:='140 - Automaticky Rezim - zasunutie pritlacenia kontaktov testera';
			SC_P4_FunkcnyTestB.IdleTime.PT:= T#1s;
			SC_P4_FunkcnyTestB.AlarmTime.PT:= T#5s;

			P4_FunkcnyTestB.OUT.KontaktyTestera_VYSUN:= FALSE;
			SC_P4_FunkcnyTestB.IdleTime.IN:= TRUE;

			IF SC_P4_FunkcnyTestB.IdleTime.Q THEN
				SC_P4_FunkcnyTestB.ResetStep:= TRUE;
				SC_P4_FunkcnyTestB.Step:= 143;
			END_IF

		143:
			SC_P4_FunkcnyTestB.StepName:='143 - Automaticky Rezim - zasunutie spodnych kontaktov';
			SC_P4_FunkcnyTestB.IdleTime.PT:= T#200ms;
			SC_P4_FunkcnyTestB.AlarmTime.PT:= T#5s;

			IF NOT SC_P4_FunkcnyTestB.Switch1 THEN
				SpodneKontakty_ZASUN:= TRUE;
				P4_FunkcnyTestB.OUT.PritlakPowerCP_VYSUN:= TRUE;
				SC_P4_FunkcnyTestB.Switch1:= TRUE;
			END_IF

			IF P4_FunkcnyTestB.IN.SpodneKontakty_ZASUNUTE THEN
				SC_P4_FunkcnyTestB.ResetStep:= TRUE;
				SC_P4_FunkcnyTestB.Step:= 145;
			END_IF

		145:
			SC_P4_FunkcnyTestB.StepName:='145 - Automaticky Rezim - zasunutie hornych kontaktov';
			SC_P4_FunkcnyTestB.IdleTime.PT:= T#200ms;
			SC_P4_FunkcnyTestB.AlarmTime.PT:= T#5s;

			IF NOT SC_P4_FunkcnyTestB.Switch1 THEN
				HorneKontakty_ZASUN:= TRUE;
				SC_P4_FunkcnyTestB.Switch1:= TRUE;
			END_IF

			IF P4_FunkcnyTestB.IN.HorneKontakty_ZASUNUTE THEN
				P4_FunkcnyTestB.OUT.PritlakPowerCP_VYSUN:= FALSE;
				SC_P4_FunkcnyTestB.ResetStep:= TRUE;
				SC_P4_FunkcnyTestB.Step:= 148;
			END_IF

		148:
			SC_P4_FunkcnyTestB.StepName:='148 - Automaticky Rezim - zasunutie pruzenia hornych kontaktov';
			SC_P4_FunkcnyTestB.IdleTime.PT:= T#500ms;
			SC_P4_FunkcnyTestB.AlarmTime.PT:= T#5s;

			IF NOT SC_P4_FunkcnyTestB.Switch1 THEN
				P4_FunkcnyTestB.OUT.OdpruzHornychKontaktov_VYSUN:= FALSE;
				P4_FunkcnyTestB.OUT.OdpruzHornychKontaktov_ZASUN:= TRUE;
				SC_P4_FunkcnyTestB.IdleTime.IN:= TRUE;
			END_IF

			IF SC_P4_FunkcnyTestB.IdleTime.Q THEN
				SC_P4_FunkcnyTestB.ResetStep:= TRUE;
				SC_P4_FunkcnyTestB.Step:= 150;
			END_IF

		150:
			SC_P4_FunkcnyTestB.StepName:='150 - Automaticky Rezim - odcentrovanie paletky';
			SC_P4_FunkcnyTestB.IdleTime.PT:= T#200ms;
			SC_P4_FunkcnyTestB.AlarmTime.PT:= T#5s;

			IF NOT SC_P4_FunkcnyTestB.Switch1 THEN
				Centrovacku_ZASUN:= TRUE;
				SC_P4_FunkcnyTestB.Switch1:= TRUE;
			END_IF

			IF P4_FunkcnyTestB.IN.Centrovanie_ZASUNUTE THEN
				IF P4_FunkcnyTestB.Manual THEN
					P4_FunkcnyTestB.STAV.RR_SekvenciaTestera_BUSY:= FALSE;
					SC_P4_FunkcnyTestB.ResetStep:= TRUE;
					SC_P4_FunkcnyTestB.Step:= 700;
				ELSE
					SC_P4_FunkcnyTestB.ResetStep:= TRUE;
					SC_P4_FunkcnyTestB.Step:= 560;
				END_IF
			END_IF

		//***************************Vyvezenie paletky**********************************************//
		560:
			SC_P4_FunkcnyTestB.StepName:='560 - Automaticky Rezim - cakam na vyvezenie na zdvižku za Funkcnym Testom B';
			SC_P4_FunkcnyTestB.IdleTime.PT:= T#200ms;
			SC_P4_FunkcnyTestB.AlarmTime.PT:= T#5s;

			IF P4_FunkcnyTestB.KoniecCyklu THEN
				SC_P4_FunkcnyTestB.ResetStep:= TRUE;
				SC_P4_FunkcnyTestB.Step:= 0;
			ELSIF NOT P4_ZdvizkaZaFunkcTestB.IN.PritomnostPaletky AND
				SC_P4_ZdvizkaZaFunkcTestB.Step = 100 AND
				NOT P4_FunkcnyTestB.STAV.PrebiehaVyvezeniePaletky AND
				P4_ZdvizkaZaFunkcTestA.STAV.PoINIT AND
				P4_ZdvizkaZaFunkcTestB.IN.Zdvizka_StrednaPoloha AND
				P4_ZdvizkaZaFunkcTestB.STAV.PoINIT THEN
				P4_FunkcnyTestB.OUT.ZasunStoper:= TRUE;
				P4_FunkcnyTestB.STAV.PrebiehaVyvezeniePaletky:= TRUE;
				SC_P4_FunkcnyTestB.ResetStep:= TRUE;
				SC_P4_FunkcnyTestB.Step:= 561;
			END_IF

		561:
			SC_P4_FunkcnyTestB.StepName:='561 - Automaticky Rezim - ukoncenie vyvazania na zdvižku za Funkcnym Testom B';
			SC_P4_FunkcnyTestB.IdleTime.PT:= T#200ms;
			SC_P4_FunkcnyTestB.AlarmTime.PT:= T#10s;

			SC_P4_FunkcnyTestB.AlarmTime.IN:= P4_FunkcnyTestB.RFID_hlava.PritomnostPaletky;
			SC_P4_FunkcnyTestB.IdleTime.IN:= NOT P4_FunkcnyTestB.RFID_hlava.PritomnostPaletky;

			IF NOT P4_FunkcnyTestB.RFID_hlava.PritomnostPaletky THEN
				TestovaciKus:= FALSE;
				Paletka[i].PAR.StavPowerCP:= '';
				Paletka[i].STAV.Komunikacia_DONE:= FALSE;
				Paletka[i].STAV.OdoslanieFotiek_DONE:= FALSE;
				P4_FunkcnyTestB.OUT.ZasunStoper:= FALSE;
				SC_P4_FunkcnyTestB.ResetStep:= TRUE;
				SC_P4_FunkcnyTestB.Step:= 100;
			ELSIF SC_P4_FunkcnyTestB.AlarmTime.Q THEN
				P34_Alarmy[451]:= TRUE;
				P4_Pracovisko.STAV.Porucha_ST2:= TRUE;
			END_IF

			//*******************************************************Manuálny režim*******************************************************************************//
		700:
			SC_P4_FunkcnyTestB.StepName:='700 - Manualny Rezim';
			SC_P4_FunkcnyTestB.IdleTime.PT:= T#8s;
			SC_P4_FunkcnyTestB.AlarmTime.PT:= T#5s;

			//Sekvencia zatvárania testera//
			IF P4_FunkcnyTestB.CMD.RR_ZatvorTester THEN
				P4_FunkcnyTestB.STAV.RR_SekvenciaTestera_BUSY:= TRUE;
				SC_P4_FunkcnyTestB.ResetStep:= TRUE;
				SC_P4_FunkcnyTestB.Step:= 110;
			END_IF

			//Ovládanie zdvižky//
			IF P4_FunkcnyTestB.CMD.RR_VysunCentrovanie THEN
				P4_FunkcnyTestB.OUT.Centrovanie_VYSUN:= TRUE;
				P4_FunkcnyTestB.OUT.Centrovanie_ZASUN:= FALSE;
			ELSE
				P4_FunkcnyTestB.OUT.Centrovanie_VYSUN:= FALSE;
				P4_FunkcnyTestB.OUT.Centrovanie_ZASUN:= TRUE;
			END_IF

			//Ovládanie pruženia horných kontaktov//
			IF P4_FunkcnyTestB.CMD.RR_VysunPruzenieKontaktov THEN
				P4_FunkcnyTestB.OUT.OdpruzHornychKontaktov_ZASUN:= FALSE;
				P4_FunkcnyTestB.OUT.OdpruzHornychKontaktov_VYSUN:= TRUE;
			ELSE
				P4_FunkcnyTestB.OUT.OdpruzHornychKontaktov_ZASUN:= TRUE;
				P4_FunkcnyTestB.OUT.OdpruzHornychKontaktov_VYSUN:= FALSE;
			END_IF

	END_CASE

END_PROGRAM

PROGRAM _EXIT
	(* Insert code here *)

END_PROGRAM
```

#### Variables.var - Local variables
```iecst
VAR
	SC_OvlCentrovacky : SequenceControlTyp;
	Centrovacku_VYSUN : BOOL;
	Centrovacku_ZASUN : BOOL;
	SC_OvlSpodnychKontaktov : SequenceControlTyp;
	SpodneKontakty_VYSUN : BOOL;
	SpodneKontakty_ZASUN : BOOL;
	SC_OvlHornychKontaktov : SequenceControlTyp;
	HorneKontakty_VYSUN : BOOL;
	HorneKontakty_ZASUN : BOOL;
	i : USINT;
	TestovaciKus : BOOL := 0;
	SC_OvlTesteraFT : SequenceControlTyp;
	SKTcpClientTester_0 : SKTcpClientTester;
	dataStr : STRING[32];
	PocetDopytovNaTester : USINT := 0;
	Cas_FunkcnyTestB : TON;
	NameranyCasFunkcnehoTestuB : TIME := T#0S;
END_VAR
```

#### IOLinkKomunikacia.st
```iecst
ACTION IOLinkKomunikacia:

	//RFID snímač paletky//
	P4_FunkcnyTestB.RFID_hlava();

END_ACTION
```

#### OvlCentrovacky.st
```iecst
ACTION OvlCentrovacky:

	//Volanie funkcie SequenceControl//
	SequenceControl(SC:= SC_OvlCentrovacky);

	CASE SC_OvlCentrovacky.Step OF

		0:
			SC_OvlCentrovacky.StepName:= '0 - Nulovanie';
			Centrovacku_VYSUN:= FALSE;
			Centrovacku_ZASUN:= FALSE;

			IF SC_P4_FunkcnyTestB.Step <> 0 THEN
				SC_OvlCentrovacky.ResetStep:= TRUE;
				SC_OvlCentrovacky.Step:= 1;
			END_IF

		1:
			SC_OvlCentrovacky.StepName:= '1 - Rozhodnutie o cinnosti';
			IF Centrovacku_VYSUN THEN
				SC_OvlCentrovacky.Step:= 10;
			ELSIF Centrovacku_ZASUN THEN
				SC_OvlCentrovacky.Step:= 20;
			END_IF

		10:
			SC_OvlCentrovacky.StepName:= '10 - Vysunutie centrovacky';
			SC_OvlCentrovacky.IdleTime.PT:= T#3s;
			SC_OvlCentrovacky.AlarmTime.PT:= T#6s;

			IF P4_FunkcnyTestB.Automat THEN
				SC_OvlCentrovacky.AlarmTime.IN:= TRUE;
			ELSE
				SC_OvlCentrovacky.IdleTime.IN:= TRUE;
			END_IF

			IF NOT SC_OvlCentrovacky.Switch1 THEN
				P4_FunkcnyTestB.OUT.Centrovanie_ZASUN:= FALSE;
                P4_FunkcnyTestB.OUT.Centrovanie_VYSUN:= TRUE;
				SC_OvlCentrovacky.Switch1:= TRUE;
			END_IF

			IF P4_FunkcnyTestB.IN.Centrovanie_VYSUNUTE OR SC_OvlCentrovacky.IdleTime.Q THEN
				SC_OvlCentrovacky.ResetStep:= TRUE;
				SC_OvlCentrovacky.Step:= 0;
			ELSIF SC_OvlCentrovacky.AlarmTime.Q THEN
				P34_Alarmy[402]:= TRUE;
				P4_Pracovisko.STAV.Porucha_ST2:= TRUE;
			END_IF

		20:
			SC_OvlCentrovacky.StepName:= '20 - Zasunutie centrovacky';
			SC_OvlCentrovacky.IdleTime.PT:= T#3s;
			SC_OvlCentrovacky.AlarmTime.PT:= T#6s;

			IF P4_FunkcnyTestB.Automat THEN
				SC_OvlCentrovacky.AlarmTime.IN:= TRUE;
			ELSE
				SC_OvlCentrovacky.IdleTime.IN:= TRUE;
			END_IF

			IF NOT SC_OvlCentrovacky.Switch1 THEN
				P4_FunkcnyTestB.OUT.Centrovanie_VYSUN:= FALSE;
                P4_FunkcnyTestB.OUT.Centrovanie_ZASUN:= TRUE;
				SC_OvlCentrovacky.Switch1:= TRUE;
			END_IF

			IF P4_FunkcnyTestB.IN.Centrovanie_ZASUNUTE OR SC_OvlCentrovacky.IdleTime.Q THEN
				SC_OvlCentrovacky.ResetStep:= TRUE;
				SC_OvlCentrovacky.Step:= 0;
			ELSIF SC_OvlCentrovacky.AlarmTime.Q THEN
				P34_Alarmy[403]:= TRUE;
				P4_Pracovisko.STAV.Porucha_ST2:= TRUE;
			END_IF

	END_CASE

END_ACTION
```

#### OvlSpodnychKontaktov.st
```iecst
ACTION OvlSpodnychKontaktov:

	//Volanie funkcie SequenceControl//
	SequenceControl(SC:= SC_OvlSpodnychKontaktov);

	CASE SC_OvlSpodnychKontaktov.Step OF

		0:
			SC_OvlSpodnychKontaktov.StepName:= '0 - Nulovanie';
			SpodneKontakty_VYSUN:= FALSE;
			SpodneKontakty_ZASUN:= FALSE;

			IF SC_P4_FunkcnyTestB.Step <> 0 THEN
				SC_OvlSpodnychKontaktov.ResetStep:= TRUE;
				SC_OvlSpodnychKontaktov.Step:= 1;
			END_IF

		1:
			SC_OvlSpodnychKontaktov.StepName:= '1 - Rozhodnutie o cinnosti';
			IF SpodneKontakty_VYSUN THEN
				SC_OvlSpodnychKontaktov.Step:= 10;
			ELSIF SpodneKontakty_ZASUN THEN
				SC_OvlSpodnychKontaktov.Step:= 20;
			END_IF

		10:
			SC_OvlSpodnychKontaktov.StepName:= '10 - Vysunutie spodnych kontaktov';
			SC_OvlSpodnychKontaktov.IdleTime.PT:= T#3s;
			SC_OvlSpodnychKontaktov.AlarmTime.PT:= T#6s;

			IF P4_FunkcnyTestB.Automat THEN
				SC_OvlSpodnychKontaktov.AlarmTime.IN:= TRUE;
			ELSE
				SC_OvlSpodnychKontaktov.IdleTime.IN:= TRUE;
			END_IF

			IF NOT SC_OvlSpodnychKontaktov.Switch1 THEN
				P4_FunkcnyTestB.OUT.SpodneKontakty_ZASUN:= FALSE;
                P4_FunkcnyTestB.OUT.SpodneKontakty_VYSUN:= TRUE;
				SC_OvlSpodnychKontaktov.Switch1:= TRUE;
			END_IF

			IF P4_FunkcnyTestB.IN.SpodneKontakty_VYSUNUTE OR SC_OvlSpodnychKontaktov.IdleTime.Q THEN
				SC_OvlSpodnychKontaktov.ResetStep:= TRUE;
				SC_OvlSpodnychKontaktov.Step:= 0;
			ELSIF SC_OvlSpodnychKontaktov.AlarmTime.Q THEN
				P34_Alarmy[425]:= TRUE;
				P4_Pracovisko.STAV.Porucha_ST2:= TRUE;
			END_IF

		20:
			SC_OvlSpodnychKontaktov.StepName:= '20 - Zasunutie spodnych kontaktov';
			SC_OvlSpodnychKontaktov.IdleTime.PT:= T#3s;
			SC_OvlSpodnychKontaktov.AlarmTime.PT:= T#6s;

			IF P4_FunkcnyTestB.Automat THEN
				SC_OvlSpodnychKontaktov.AlarmTime.IN:= TRUE;
			ELSE
				SC_OvlSpodnychKontaktov.IdleTime.IN:= TRUE;
			END_IF

			IF NOT SC_OvlSpodnychKontaktov.Switch1 THEN
				P4_FunkcnyTestB.OUT.SpodneKontakty_VYSUN:= FALSE;
                P4_FunkcnyTestB.OUT.SpodneKontakty_ZASUN:= TRUE;
				SC_OvlSpodnychKontaktov.Switch1:= TRUE;
			END_IF

			IF P4_FunkcnyTestB.IN.SpodneKontakty_ZASUNUTE OR SC_OvlSpodnychKontaktov.IdleTime.Q THEN
				SC_OvlSpodnychKontaktov.ResetStep:= TRUE;
				SC_OvlSpodnychKontaktov.Step:= 0;
			ELSIF SC_OvlSpodnychKontaktov.AlarmTime.Q THEN
				P34_Alarmy[426]:= TRUE;
				P4_Pracovisko.STAV.Porucha_ST2:= TRUE;
			END_IF

	END_CASE

END_ACTION
```

#### OvlHornychKontaktov.st
```iecst
ACTION OvlHornychKontaktov:

	//Volanie funkcie SequenceControl//
	SequenceControl(SC:= SC_OvlHornychKontaktov);

	CASE SC_OvlHornychKontaktov.Step OF

		0:
			SC_OvlHornychKontaktov.StepName:= '0 - Nulovanie';
			HorneKontakty_VYSUN:= FALSE;
			HorneKontakty_ZASUN:= FALSE;

			IF SC_P4_FunkcnyTestB.Step <> 0 THEN
				SC_OvlHornychKontaktov.ResetStep:= TRUE;
				SC_OvlHornychKontaktov.Step:= 1;
			END_IF

		1:
			SC_OvlHornychKontaktov.StepName:= '1 - Rozhodnutie o cinnosti';
			IF HorneKontakty_VYSUN THEN
				SC_OvlHornychKontaktov.Step:= 10;
			ELSIF HorneKontakty_ZASUN THEN
				SC_OvlHornychKontaktov.Step:= 20;
			END_IF

		10:
			SC_OvlHornychKontaktov.StepName:= '10 - Vysunutie hornych kontaktov';
			SC_OvlHornychKontaktov.IdleTime.PT:= T#3s;
			SC_OvlHornychKontaktov.AlarmTime.PT:= T#6s;

			IF P4_FunkcnyTestB.Automat THEN
				SC_OvlHornychKontaktov.AlarmTime.IN:= TRUE;
			ELSE
				SC_OvlHornychKontaktov.IdleTime.IN:= TRUE;
			END_IF

			IF NOT SC_OvlHornychKontaktov.Switch1 THEN
				P4_FunkcnyTestB.OUT.HorneKontakty_ZASUN:= FALSE;
				P4_FunkcnyTestB.OUT.HorneKontakty_VYSUN:= TRUE;
				SC_OvlHornychKontaktov.Switch1:= TRUE;
			END_IF

			IF P4_FunkcnyTestB.IN.HorneKontakty_VYSUNUTE OR SC_OvlHornychKontaktov.IdleTime.Q THEN
				SC_OvlHornychKontaktov.ResetStep:= TRUE;
				SC_OvlHornychKontaktov.Step:= 0;
			ELSIF SC_OvlHornychKontaktov.AlarmTime.Q THEN
				P34_Alarmy[423]:= TRUE;
				P4_Pracovisko.STAV.Porucha_ST2:= TRUE;
			END_IF

		20:
			SC_OvlHornychKontaktov.StepName:= '20 - Zasunutie hornych kontaktov';
			SC_OvlHornychKontaktov.IdleTime.PT:= T#3s;
			SC_OvlHornychKontaktov.AlarmTime.PT:= T#6s;

			IF P4_FunkcnyTestB.Automat THEN
				SC_OvlHornychKontaktov.AlarmTime.IN:= TRUE;
			ELSE
				SC_OvlHornychKontaktov.IdleTime.IN:= TRUE;
			END_IF

			IF NOT SC_OvlHornychKontaktov.Switch1 THEN
				P4_FunkcnyTestB.OUT.HorneKontakty_VYSUN:= FALSE;
				P4_FunkcnyTestB.OUT.HorneKontakty_ZASUN:= TRUE;
				SC_OvlHornychKontaktov.Switch1:= TRUE;
			END_IF

			IF P4_FunkcnyTestB.IN.HorneKontakty_ZASUNUTE OR SC_OvlHornychKontaktov.IdleTime.Q THEN
				SC_OvlHornychKontaktov.ResetStep:= TRUE;
				SC_OvlHornychKontaktov.Step:= 0;
			ELSIF SC_OvlHornychKontaktov.AlarmTime.Q THEN
				P34_Alarmy[424]:= TRUE;
				P4_Pracovisko.STAV.Porucha_ST2:= TRUE;
			END_IF

	END_CASE

END_ACTION
```

#### COM_Tester.st
```iecst
ACTION COM_Tester:

		//Parametre komunikácie//
    memcpy(ADR(SKTcpClientTester_0.Params.IPaddrServ),ADR('192.168.128.252'),SIZEOF('192.168.128.252'));
    SKTcpClientTester_0.Params.IPportClient := P4_FunkcnyTestB.PAR.CisloPortuKlienta;
    SKTcpClientTester_0.Params.IPportServ := 1030;
    SKTcpClientTester_0.Params.RecvTimeout := 10000;
    strcpy(ADR(SKTcpClientTester_0.Params.Packet.data),ADR(dataStr));
    SKTcpClientTester_0();

    Cas_FunkcnyTestB.PT:= T#1M;
    Cas_FunkcnyTestB();

    //Volanie funkcie SequenceControl//
    SequenceControl(SC:= SC_OvlTesteraFT);

    CASE SC_OvlTesteraFT.Step OF

        0:
            SC_OvlTesteraFT.StepName:= '0 - Nulovanie';
            SKTcpClientTester_0.Enable:= TRUE;
            SKTcpClientTester_0.Cmd.Send:= FALSE;
			P4_FunkcnyTestB.STAV.TestovanieUkoncene:= FALSE;
			P4_FunkcnyTestB.STAV.TesterNeodpoveda:= FALSE;
            PocetDopytovNaTester:= 0;
            SC_OvlTesteraFT.ResetStep:= TRUE;
            SC_OvlTesteraFT.Step:= 1;

        1:
            SC_OvlTesteraFT.StepName:= '1 - Cakam na spustenie testera';
            IF P4_FunkcnyTestB.CMD.StartTestovania THEN
                P4_FunkcnyTestB.STAV.Vysledok_FV_Testu:= '';
                Cas_FunkcnyTestB.IN:= TRUE;
                NameranyCasFunkcnehoTestuB:= 0;
                SC_OvlTesteraFT.Step:= 10;
            END_IF

        10:
            SC_OvlTesteraFT.StepName:= '10 - Dopyt na stav testera - typ 0';
            SC_OvlTesteraFT.IdleTime.PT:= T#300ms;
            SC_OvlTesteraFT.AlarmTime.PT:= T#10s;
            SC_OvlTesteraFT.IdleTime.IN:= TRUE;
            SC_OvlTesteraFT.AlarmTime.IN:= TRUE;

            SKTcpClientTester_0.Params.Packet.type:= 0;
            SKTcpClientTester_0.Params.Packet.workplace:= 49;
            SKTcpClientTester_0.Params.Packet.id:= 2;
            SKTcpClientTester_0.Cmd.Close:= FALSE;
			SKTcpClientTester_0.Cmd.Send:= TRUE;

            IF SKTcpClientTester_0.Cmd.Send AND NOT SKTcpClientTester_0.Status.staReceived AND NOT SKTcpClientTester_0.Status.staError THEN
                SC_OvlTesteraFT.ResetStep:= TRUE;
                SC_OvlTesteraFT.Step:= 13;
            ELSIF SC_OvlTesteraFT.AlarmTime.Q AND (SKTcpClientTester_0.Status.staReceived OR SKTcpClientTester_0.Status.staError) THEN
                PocetDopytovNaTester:= PocetDopytovNaTester + 1;
				SKTcpClientTester_0.Cmd.Send:= FALSE;
				SKTcpClientTester_0.Cmd.Close:= TRUE;
				SC_OvlTesteraFT.ResetStep:= TRUE;
                SC_OvlTesteraFT.Step:= 12;
            END_IF

        12:
            SC_OvlTesteraFT.StepName:= '12 - Dopyt na stav testera - cakam na opatovny dopyt na tester';
            SC_OvlTesteraFT.IdleTime.PT:= T#800ms;
            SC_OvlTesteraFT.AlarmTime.PT:= T#5s;
            SC_OvlTesteraFT.IdleTime.IN:= TRUE;
            SKTcpClientTester_0.Cmd.Send:= FALSE;

            IF PocetDopytovNaTester < 10 THEN
                IF SC_OvlTesteraFT.IdleTime.Q THEN
                    SC_OvlTesteraFT.ResetStep:= TRUE;
                    SC_OvlTesteraFT.Step:= 10;
                END_IF
            ELSE
                P4_FunkcnyTestB.STAV.Vysledok_FV_Testu:= 'NG';
                P4_FunkcnyTestB.STAV.TesterNeodpoveda:= TRUE;
                SC_OvlTesteraFT.ResetStep:= TRUE;
                SC_OvlTesteraFT.Step:= 100;
            END_IF

        13:
            SC_OvlTesteraFT.StepName:= '13 - Odpoved na stav testera - typ 0';
            SC_OvlTesteraFT.IdleTime.PT:= T#800ms;
            SC_OvlTesteraFT.AlarmTime.PT:= T#10s;
            SC_OvlTesteraFT.IdleTime.IN:= TRUE;

            IF SKTcpClientTester_0.Status.staReceived AND SKTcpClientTester_0.Status.DataRecv[2]= 0 AND SKTcpClientTester_0.Status.DataRecv[5]= 2 THEN
                SKTcpClientTester_0.Cmd.Send:= FALSE;
                SC_OvlTesteraFT.ResetStep:= TRUE;
                SC_OvlTesteraFT.Step:= 15;
            ELSIF SKTcpClientTester_0.Status.staReceived AND SKTcpClientTester_0.Status.DataRecv[2]= 0 AND SKTcpClientTester_0.Status.DataRecv[5]= 1 THEN
                SKTcpClientTester_0.Cmd.Send:= FALSE;
                SKTcpClientTester_0.Cmd.Close:= TRUE;
				IF SC_OvlTesteraFT.IdleTime.Q THEN
                    SC_OvlTesteraFT.ResetStep:= TRUE;
                    SC_OvlTesteraFT.Step:= 10;
                END_IF
            ELSIF SKTcpClientTester_0.Status.staReceived AND SKTcpClientTester_0.Status.DataRecv[2]= 0 AND SKTcpClientTester_0.Status.DataRecv[5]= 0 THEN
                SKTcpClientTester_0.Cmd.Send:= FALSE;
                SKTcpClientTester_0.Cmd.Close:= TRUE;
				IF SC_OvlTesteraFT.IdleTime.Q THEN
                    SC_OvlTesteraFT.ResetStep:= TRUE;
                    SC_OvlTesteraFT.Step:= 10;
                END_IF
            ELSIF SKTcpClientTester_0.Status.staError THEN
                SKTcpClientTester_0.Cmd.Send:= FALSE;
                P4_FunkcnyTestB.STAV.Vysledok_FV_Testu:= 'NG';
                P4_FunkcnyTestB.STAV.TesterNeodpoveda:= TRUE;
                SC_OvlTesteraFT.ResetStep:= TRUE;
                SC_OvlTesteraFT.Step:= 100;
            END_IF

        15:
            SC_OvlTesteraFT.StepName:= '15 - Poslanie QR kodu Power CP - typ 1';
            SC_OvlTesteraFT.IdleTime.PT:= T#300ms;
            SC_OvlTesteraFT.AlarmTime.PT:= T#10s;
            SC_OvlTesteraFT.IdleTime.IN:= TRUE;

            SKTcpClientTester_0.Params.Packet.type:= 1;
            SKTcpClientTester_0.Params.Packet.workplace:= 49;
            SKTcpClientTester_0.Params.Packet.id:= 2;
			dataStr:= Paletka[i].PAR.QRkodPowerCP;
		    SKTcpClientTester_0.Cmd.Send:= TRUE;

            IF SKTcpClientTester_0.Cmd.Send AND NOT SKTcpClientTester_0.Status.staReceived AND NOT SKTcpClientTester_0.Status.staError THEN
                SC_OvlTesteraFT.ResetStep:= TRUE;
                SC_OvlTesteraFT.Step:= 18;
            END_IF

        18:
            SC_OvlTesteraFT.StepName:= '18 - Odpoved na poslanie QR kodu - typ 1';
            SC_OvlTesteraFT.IdleTime.PT:= T#300ms;
            SC_OvlTesteraFT.AlarmTime.PT:= T#10s;
            SC_OvlTesteraFT.IdleTime.IN:= TRUE;

            IF SKTcpClientTester_0.Status.staReceived AND SKTcpClientTester_0.Status.DataRecv[2]= 1 AND SKTcpClientTester_0.Status.DataRecv[5]= 0 THEN
                SKTcpClientTester_0.Cmd.Send:= FALSE;
                SC_OvlTesteraFT.ResetStep:= TRUE;
                SC_OvlTesteraFT.Step:= 20;
            ELSIF SKTcpClientTester_0.Status.staReceived AND SKTcpClientTester_0.Status.DataRecv[2]= 1 AND SKTcpClientTester_0.Status.DataRecv[5]= 2 THEN
                SKTcpClientTester_0.Cmd.Send:= FALSE;
                IF SC_OvlTesteraFT.IdleTime.Q THEN
                    SC_OvlTesteraFT.ResetStep:= TRUE;
                    SC_OvlTesteraFT.Step:= 15;
                END_IF
            ELSIF SKTcpClientTester_0.Status.staReceived AND SKTcpClientTester_0.Status.DataRecv[2]= 1 AND SKTcpClientTester_0.Status.DataRecv[5]= 1 THEN
                SKTcpClientTester_0.Cmd.Send:= FALSE;
                P4_FunkcnyTestB.STAV.Vysledok_FV_Testu:= 'NG';
                P4_FunkcnyTestB.STAV.TestovanieUkoncene:= TRUE;
                SC_OvlTesteraFT.ResetStep:= TRUE;
                SC_OvlTesteraFT.Step:= 100;
            ELSIF SKTcpClientTester_0.Status.staError THEN
                SKTcpClientTester_0.Cmd.Send:= FALSE;
                P4_FunkcnyTestB.STAV.Vysledok_FV_Testu:= 'NG';
                P4_FunkcnyTestB.STAV.TesterNeodpoveda:= TRUE;
                SC_OvlTesteraFT.ResetStep:= TRUE;
                SC_OvlTesteraFT.Step:= 100;
            END_IF

        20:
            SC_OvlTesteraFT.StepName:= '20 - Dopyt na stav testera - typ 0';
            SC_OvlTesteraFT.IdleTime.PT:= T#300ms;
            SC_OvlTesteraFT.AlarmTime.PT:= T#10s;
            SC_OvlTesteraFT.IdleTime.IN:= TRUE;

            SKTcpClientTester_0.Params.Packet.type:= 0;
            SKTcpClientTester_0.Params.Packet.workplace:= 49;
            SKTcpClientTester_0.Params.Packet.id:= 2;
            SKTcpClientTester_0.Cmd.Send:= TRUE;

            IF SKTcpClientTester_0.Cmd.Send AND NOT SKTcpClientTester_0.Status.staReceived AND NOT SKTcpClientTester_0.Status.staError THEN
                SC_OvlTesteraFT.ResetStep:= TRUE;
                SC_OvlTesteraFT.Step:= 23;
            END_IF

        23:
            SC_OvlTesteraFT.StepName:= '23 - Odpoved na stav testera - typ 0';
            SC_OvlTesteraFT.IdleTime.PT:= T#300ms;
            SC_OvlTesteraFT.AlarmTime.PT:= T#10s;
            SC_OvlTesteraFT.IdleTime.IN:= TRUE;

            IF SKTcpClientTester_0.Status.staReceived AND SKTcpClientTester_0.Status.DataRecv[2]= 0 AND SKTcpClientTester_0.Status.DataRecv[5]= 3 THEN
                SKTcpClientTester_0.Cmd.Send:= FALSE;
                IF SC_OvlTesteraFT.IdleTime.Q THEN
                    SC_OvlTesteraFT.ResetStep:= TRUE;
                    SC_OvlTesteraFT.Step:= 20;
                END_IF
            ELSIF SKTcpClientTester_0.Status.staReceived AND SKTcpClientTester_0.Status.DataRecv[2]= 0 AND SKTcpClientTester_0.Status.DataRecv[5]= 4 THEN
                SKTcpClientTester_0.Cmd.Send:= FALSE;
                SC_OvlTesteraFT.ResetStep:= TRUE;
                SC_OvlTesteraFT.Step:= 25;
            ELSIF SKTcpClientTester_0.Status.staReceived AND SKTcpClientTester_0.Status.DataRecv[2]= 0 AND SKTcpClientTester_0.Status.DataRecv[5]= 0 THEN
                SKTcpClientTester_0.Cmd.Send:= FALSE;
                P4_FunkcnyTestB.STAV.Vysledok_FV_Testu:= 'NG';
                P4_FunkcnyTestB.STAV.TestovanieUkoncene:= TRUE;
                SC_OvlTesteraFT.ResetStep:= TRUE;
                SC_OvlTesteraFT.Step:= 100;
            ELSIF SKTcpClientTester_0.Status.staError THEN
                SKTcpClientTester_0.Cmd.Send:= FALSE;
                P4_FunkcnyTestB.STAV.Vysledok_FV_Testu:= 'NG';
                P4_FunkcnyTestB.STAV.TesterNeodpoveda:= TRUE;
                SC_OvlTesteraFT.ResetStep:= TRUE;
                SC_OvlTesteraFT.Step:= 100;
            END_IF

        25:
            SC_OvlTesteraFT.StepName:= '25 - Dopyt na vysledok testu - typ 2';
            SC_OvlTesteraFT.IdleTime.PT:= T#300ms;
            SC_OvlTesteraFT.AlarmTime.PT:= T#10s;
            SC_OvlTesteraFT.IdleTime.IN:= TRUE;

            SKTcpClientTester_0.Params.Packet.type:= 2;
            SKTcpClientTester_0.Params.Packet.workplace:= 49;
            SKTcpClientTester_0.Params.Packet.id:= 2;
            SKTcpClientTester_0.Cmd.Send:= TRUE;

            IF SKTcpClientTester_0.Cmd.Send AND NOT SKTcpClientTester_0.Status.staReceived AND NOT SKTcpClientTester_0.Status.staError THEN
                SC_OvlTesteraFT.ResetStep:= TRUE;
                SC_OvlTesteraFT.Step:= 28;
            END_IF

        28:
            SC_OvlTesteraFT.StepName:= '28 - Odpoved na vysledok testu - typ 2';
            SC_OvlTesteraFT.IdleTime.PT:= T#300ms;
            SC_OvlTesteraFT.AlarmTime.PT:= T#10s;
            SC_OvlTesteraFT.IdleTime.IN:= TRUE;

            IF SKTcpClientTester_0.Status.staReceived AND SKTcpClientTester_0.Status.DataRecv[2]= 2 AND SKTcpClientTester_0.Status.DataRecv[5]= 1 THEN
                SKTcpClientTester_0.Cmd.Send:= FALSE;
                P4_FunkcnyTestB.STAV.Vysledok_FV_Testu:= 'OK';
                SC_OvlTesteraFT.ResetStep:= TRUE;
                SC_OvlTesteraFT.Step:= 30;
            ELSIF SKTcpClientTester_0.Status.staReceived AND SKTcpClientTester_0.Status.DataRecv[2]= 2 AND SKTcpClientTester_0.Status.DataRecv[5]= 2 THEN
                SKTcpClientTester_0.Cmd.Send:= FALSE;
                P4_FunkcnyTestB.STAV.Vysledok_FV_Testu:= 'NG';
                SC_OvlTesteraFT.ResetStep:= TRUE;
                SC_OvlTesteraFT.Step:= 30;
            ELSIF SKTcpClientTester_0.Status.staReceived AND SKTcpClientTester_0.Status.DataRecv[2]= 2 AND SKTcpClientTester_0.Status.DataRecv[5]= 0 THEN
                SKTcpClientTester_0.Cmd.Send:= FALSE;
                IF SC_OvlTesteraFT.IdleTime.Q THEN
                    SC_OvlTesteraFT.ResetStep:= TRUE;
                    SC_OvlTesteraFT.Step:= 25;
                END_IF
            ELSIF SKTcpClientTester_0.Status.staReceived AND SKTcpClientTester_0.Status.DataRecv[2]= 2 AND SKTcpClientTester_0.Status.DataRecv[5]= 3 THEN
                SKTcpClientTester_0.Cmd.Send:= FALSE;
                IF SC_OvlTesteraFT.IdleTime.Q THEN
                    SC_OvlTesteraFT.ResetStep:= TRUE;
                    SC_OvlTesteraFT.Step:= 25;
                END_IF
            ELSIF SKTcpClientTester_0.Status.staError THEN
                SKTcpClientTester_0.Cmd.Send:= FALSE;
                P4_FunkcnyTestB.STAV.Vysledok_FV_Testu:= 'NG';
                P4_FunkcnyTestB.STAV.TesterNeodpoveda:= TRUE;
                SC_OvlTesteraFT.ResetStep:= TRUE;
                SC_OvlTesteraFT.Step:= 100;
            END_IF

        30:
            SC_OvlTesteraFT.StepName:= '30 - Potvrdenie precitanie vysledkov testu - typ 3';
            SC_OvlTesteraFT.IdleTime.PT:= T#300ms;
            SC_OvlTesteraFT.AlarmTime.PT:= T#10s;
            SC_OvlTesteraFT.IdleTime.IN:= TRUE;

            SKTcpClientTester_0.Params.Packet.type:= 3;
            SKTcpClientTester_0.Params.Packet.workplace:= 49;
            SKTcpClientTester_0.Params.Packet.id:= 2;
            SKTcpClientTester_0.Cmd.Send:= TRUE;

            IF SKTcpClientTester_0.Cmd.Send AND NOT SKTcpClientTester_0.Status.staReceived AND NOT SKTcpClientTester_0.Status.staError THEN
                SC_OvlTesteraFT.ResetStep:= TRUE;
                SC_OvlTesteraFT.Step:= 33;
            END_IF

        33:
            SC_OvlTesteraFT.StepName:= '33 - Odpoved testera na potvrdenie vysledkov - typ 3';
            SC_OvlTesteraFT.IdleTime.PT:= T#500ms;
            SC_OvlTesteraFT.AlarmTime.PT:= T#10s;

            IF SKTcpClientTester_0.Status.staReceived AND SKTcpClientTester_0.Status.DataRecv[2]= 3 AND SKTcpClientTester_0.Status.DataRecv[5]= 0 THEN
                SKTcpClientTester_0.Cmd.Send:= FALSE;
                P4_FunkcnyTestB.STAV.TestovanieUkoncene:= TRUE;
                SC_OvlTesteraFT.ResetStep:= TRUE;
                SC_OvlTesteraFT.Step:= 100;
            ELSIF SKTcpClientTester_0.Status.staReceived AND SKTcpClientTester_0.Status.DataRecv[2]= 3 AND SKTcpClientTester_0.Status.DataRecv[5]= 1 THEN
                P4_FunkcnyTestB.STAV.Vysledok_FV_Testu:= 'NG';
                P4_FunkcnyTestB.STAV.TestovanieUkoncene:= TRUE;
                SKTcpClientTester_0.Cmd.Send:= FALSE;
                SC_OvlTesteraFT.ResetStep:= TRUE;
                SC_OvlTesteraFT.Step:= 100;
            ELSIF SKTcpClientTester_0.Status.staError THEN
                SKTcpClientTester_0.Cmd.Send:= FALSE;
				P4_FunkcnyTestB.STAV.Vysledok_FV_Testu:= 'NG';
				P4_FunkcnyTestB.STAV.TesterNeodpoveda:= TRUE;
				SC_OvlTesteraFT.ResetStep:= TRUE;
                SC_OvlTesteraFT.Step:= 100;
            END_IF

        100:
            SC_OvlTesteraFT.StepName:= '100 - Cakam na zrusenie signalu start testovania';
            SC_OvlTesteraFT.IdleTime.PT:= T#3s;
            SC_OvlTesteraFT.AlarmTime.PT:= T#10s;

            NameranyCasFunkcnehoTestuB:= Cas_FunkcnyTestB.ET;
            Cas_FunkcnyTestB.IN:= FALSE;

            IF NOT P4_FunkcnyTestB.CMD.StartTestovania THEN
                SC_OvlTesteraFT.ResetStep:= TRUE;
                SC_OvlTesteraFT.Step:= 0;
            END_IF

    END_CASE

END_ACTION
```

### Program Logical/Program/Pracovisko_4/P4_ZdvizkaZaFunkcTestA (IEC)

#### Main.st - Init, cyclic, exit code
```iecst
PROGRAM _INIT
	(* Insert code here *)

END_PROGRAM

PROGRAM _CYCLIC

	//Volanie funkcie SequenceControl//
	SequenceControl(SC:= SC_P4_ZdvizkaZaFunkcTestA);

	//Volanie podprogramov//
	OvlZdvizky;

	//Reset sekcie //
	IF P4_ZdvizkaZaFunkcTestA.Reset THEN
		SC_P4_ZdvizkaZaFunkcTestA.Step:= 0;
		P4_ZdvizkaZaFunkcTestA.Reset:= FALSE;
	ELSIF NOT Safety.STAV.Linka_ZonaCS_AKTIVNA THEN
		SC_P4_ZdvizkaZaFunkcTestA.Step:= 0;
	END_IF

	CASE SC_P4_ZdvizkaZaFunkcTestA.Step OF

		0:
			SC_P4_ZdvizkaZaFunkcTestA.StepName:='0 - Nulovanie';
			SC_OvlZdvizky.Step:= 0;
			P4_ZdvizkaZaFunkcTestA.Automat:= FALSE;
			P4_ZdvizkaZaFunkcTestA.KoniecCyklu:= FALSE;
			P4_ZdvizkaZaFunkcTestA.Manual:= FALSE;
			P4_ZdvizkaZaFunkcTestA.STAV.PoINIT:= FALSE;
			P4_ZdvizkaZaFunkcTestA.OUT.TlmicPaletky_VYSUN:= FALSE;
			P4_ZdvizkaZaFunkcTestA.OUT.TlmicPaletky_ZASUN:= FALSE;

			P4_FunkcnyTestA.STAV.PrebiehaVyvezeniePaletky:= FALSE;
			P4_ZdvizkaZaFunkcTestA.STAV.PrebiehaVyvezeniePaletky:= FALSE;
			P4_ZdvizkaZaFunkcTestB.STAV.PrebiehaVyvezeniePaletky:= FALSE;

			IF Safety.STAV.Linka_ZonaCS_AKTIVNA AND
				Safety.STAV.P4_ZonaBunky_AKTIVNA AND
				P4_Pracovisko.STAV.HardwareBunky_OK AND
				NOT P3_Pracovisko.STAV.Porucha_ST1 AND
				NOT P3_Pracovisko.STAV.Porucha_ST2 AND
				NOT P3_Pracovisko.STAV.Porucha_ST3 AND
				NOT P3_Pracovisko.STAV.Porucha_ST4 AND
				NOT P3_Pracovisko.STAV.Porucha_ST5 AND
				NOT P3_Pracovisko.STAV.Porucha_ST6 AND
				NOT P3_Pracovisko.STAV.Porucha_ST7 AND
				NOT P3_Pracovisko.STAV.Porucha_ST8 THEN
				SC_P4_ZdvizkaZaFunkcTestA.ResetStep:= TRUE;
				SC_P4_ZdvizkaZaFunkcTestA.Step:= 1;
			END_IF

		1:
			SC_P4_ZdvizkaZaFunkcTestA.StepName:='1 - Cakam na spustenie vyroby';
			P4_ZdvizkaZaFunkcTestA.KoniecCyklu:= FALSE;
			IF P4_ZdvizkaZaFunkcTestA.Automat THEN
				SC_P4_ZdvizkaZaFunkcTestA.Step:= 2;
			ELSIF P4_ZdvizkaZaFunkcTestA.Manual THEN
				SC_P4_ZdvizkaZaFunkcTestA.Step:= 700;
			END_IF

			//********************************************************Inicializácia****************************************************************************//

		2:
			SC_P4_ZdvizkaZaFunkcTestA.StepName:='2 - Inicializacia - cakam na spustenie inicializacie';
			SC_P4_ZdvizkaZaFunkcTestA.IdleTime.PT:= T#500ms;
			SC_P4_ZdvizkaZaFunkcTestA.AlarmTime.PT:= T#5s;

			IF P4_Dopravniky.STAV.PoINIT THEN
				SC_P4_ZdvizkaZaFunkcTestA.ResetStep:= TRUE;
				SC_P4_ZdvizkaZaFunkcTestA.Step:= 5;
			END_IF

		5:
			SC_P4_ZdvizkaZaFunkcTestA.StepName:='5 - Inicializacia - kontrola pozicie zdvizky';
			SC_P4_ZdvizkaZaFunkcTestA.IdleTime.PT:= T#500ms;
			SC_P4_ZdvizkaZaFunkcTestA.AlarmTime.PT:= T#5s;

			IF P4_ZdvizkaZaFunkcTestA.IN.Zdvizka_StrednaPoloha AND P4_ZdvizkaZaFunkcTestA.IN.PritomnostPaletky THEN
				P4_ZdvizkaZaFunkcTestA.STAV.PoINIT:= TRUE;
				SC_P4_ZdvizkaZaFunkcTestA.ResetStep:= TRUE;
				SC_P4_ZdvizkaZaFunkcTestA.Step:= 100;
			ELSE
				SC_P4_ZdvizkaZaFunkcTestA.ResetStep:= TRUE;
				SC_P4_ZdvizkaZaFunkcTestA.Step:= 8;
			END_IF

		8:
			SC_P4_ZdvizkaZaFunkcTestA.StepName:='8 - Inicializacia - presun zdvizky do hornej polohy';
			SC_P4_ZdvizkaZaFunkcTestA.IdleTime.PT:= T#5s;
			SC_P4_ZdvizkaZaFunkcTestA.AlarmTime.PT:= T#5s;

			IF NOT SC_P4_ZdvizkaZaFunkcTestA.Switch1 AND SC_OvlZdvizky.Step = 1 THEN
				Zdvizku_VYSUN:= TRUE;
				P4_ZdvizkaZaFunkcTestA.OUT.TlmicPaletky_VYSUN:= FALSE;
				P4_ZdvizkaZaFunkcTestA.OUT.TlmicPaletky_ZASUN:= TRUE;
				SC_P4_ZdvizkaZaFunkcTestA.Switch1:= TRUE;
			END_IF

			IF P4_ZdvizkaZaFunkcTestA.IN.Zdvizka_HornaPoloha AND P4_ZdvizkaZaFunkcTestA.IN.TlmicPaletky_ZASUNUTY THEN
				SC_P4_ZdvizkaZaFunkcTestA.ResetStep:= TRUE;
				SC_P4_ZdvizkaZaFunkcTestA.Step:= 10;
			END_IF

		10:
			SC_P4_ZdvizkaZaFunkcTestA.StepName:='10 - Inicializacia - kontrola pritomnosti paletky na zdvizke za Funkcnym Testom B';
			SC_P4_ZdvizkaZaFunkcTestA.IdleTime.PT:= T#500ms;
			SC_P4_ZdvizkaZaFunkcTestA.AlarmTime.PT:= T#5s;

			IF NOT P4_ZdvizkaZaFunkcTestB.IN.PritomnostPaletky THEN
				P4_ZdvizkaZaFunkcTestB.OUT.Zdvizku_VYSUN:= TRUE;
				SC_P4_ZdvizkaZaFunkcTestA.ResetStep:= TRUE;
				SC_P4_ZdvizkaZaFunkcTestA.Step:= 11;
			ELSE
				SC_P4_ZdvizkaZaFunkcTestA.ResetStep:= TRUE;
				SC_P4_ZdvizkaZaFunkcTestA.Step:= 13;
			END_IF

		11:
			SC_P4_ZdvizkaZaFunkcTestA.StepName:='11 - Inicializacia - cakam na zodvihnutie zdvizky za Funkcnym Testom B';
			SC_P4_ZdvizkaZaFunkcTestA.IdleTime.PT:= T#500ms;
			SC_P4_ZdvizkaZaFunkcTestA.AlarmTime.PT:= T#5s;

			IF P4_ZdvizkaZaFunkcTestB.IN.Zdvizka_HornaPoloha THEN
				SC_P4_ZdvizkaZaFunkcTestA.ResetStep:= TRUE;
				SC_P4_ZdvizkaZaFunkcTestA.Step:= 13;
			END_IF

		13:
			SC_P4_ZdvizkaZaFunkcTestA.StepName:='13 - Inicializacia - spustenie priecneho dopravnika';
			SC_P4_ZdvizkaZaFunkcTestA.IdleTime.PT:= T#500ms;
			SC_P4_ZdvizkaZaFunkcTestA.AlarmTime.PT:= T#7s;

			SC_P4_ZdvizkaZaFunkcTestA.IdleTime.IN:= P4_ZdvizkaZaFunkcTestA.IN.PritomnostPaletky AND P4_ZdvizkaZaFunkcTestA.IN.PoziciaPaletky_OK;

			IF NOT SC_P4_ZdvizkaZaFunkcTestA.Switch1 THEN
				P4_Dopravniky.OUT.PriecnyDopravnik_VPRED:= TRUE;
				SC_P4_ZdvizkaZaFunkcTestA.AlarmTime.IN:= TRUE;
				SC_P4_ZdvizkaZaFunkcTestA.Switch1:= TRUE;
			END_IF

			IF SC_P4_ZdvizkaZaFunkcTestA.IdleTime.Q THEN
				P4_Dopravniky.OUT.PriecnyDopravnik_VPRED:= FALSE;
				SC_P4_ZdvizkaZaFunkcTestA.ResetStep:= TRUE;
				SC_P4_ZdvizkaZaFunkcTestA.Step:= 15;
			ELSIF SC_P4_ZdvizkaZaFunkcTestA.AlarmTime.Q THEN
				P4_Dopravniky.OUT.PriecnyDopravnik_VPRED:= FALSE;
				SC_P4_ZdvizkaZaFunkcTestA.ResetStep:= TRUE;
				SC_P4_ZdvizkaZaFunkcTestA.Step:= 15;
			END_IF

		15:
			SC_P4_ZdvizkaZaFunkcTestA.StepName:='15 - Inicializacia - presun zdvizky do strednej polohy';
			SC_P4_ZdvizkaZaFunkcTestA.IdleTime.PT:= T#500ms;
			SC_P4_ZdvizkaZaFunkcTestA.AlarmTime.PT:= T#5s;

			IF NOT SC_P4_ZdvizkaZaFunkcTestA.Switch1 AND SC_OvlZdvizky.Step = 1 THEN
				Zdvizku_VYSTRED:= TRUE;
				P4_ZdvizkaZaFunkcTestB.OUT.Zdvizku_VYSUN:= FALSE;
				SC_P4_ZdvizkaZaFunkcTestA.Switch1:= TRUE;
			END_IF

			IF P4_ZdvizkaZaFunkcTestA.IN.Zdvizka_StrednaPoloha AND P4_ZdvizkaZaFunkcTestB.IN.Zdvizka_StrednaPoloha THEN
				IF P4_ZdvizkaZaFunkcTestA.IN.PritomnostPaletky THEN
					P4_ZdvizkaZaFunkcTestA.STAV.PoINIT:= TRUE;
					SC_P4_ZdvizkaZaFunkcTestA.ResetStep:= TRUE;
					SC_P4_ZdvizkaZaFunkcTestA.Step:= 100;
				ELSE
					SC_P4_ZdvizkaZaFunkcTestA.ResetStep:= TRUE;
					SC_P4_ZdvizkaZaFunkcTestA.Step:= 18;
				END_IF
			END_IF

		18:
			SC_P4_ZdvizkaZaFunkcTestA.StepName:='18 - Inicializacia - vysunutie tlmica paletky';
			SC_P4_ZdvizkaZaFunkcTestA.IdleTime.PT:= T#1s;
			SC_P4_ZdvizkaZaFunkcTestA.AlarmTime.PT:= T#5s;

			SC_P4_ZdvizkaZaFunkcTestA.IdleTime.IN:= NOT P4_ZdvizkaZaFunkcTestA.IN.TlmicPaletky_ZASUNUTY;

			IF NOT SC_P4_ZdvizkaZaFunkcTestA.Switch1 THEN
				P4_ZdvizkaZaFunkcTestA.OUT.TlmicPaletky_ZASUN:= FALSE;
				P4_ZdvizkaZaFunkcTestA.OUT.TlmicPaletky_VYSUN:= TRUE;
				SC_P4_ZdvizkaZaFunkcTestA.Switch1:= TRUE;
			END_IF

			IF SC_P4_ZdvizkaZaFunkcTestA.IdleTime.Q THEN
				P4_ZdvizkaZaFunkcTestA.OUT.TlmicPaletky_ZASUN:= FALSE;
				P4_ZdvizkaZaFunkcTestA.OUT.TlmicPaletky_VYSUN:= FALSE;
				P4_ZdvizkaZaFunkcTestA.STAV.PoINIT:= TRUE;
				SC_P4_ZdvizkaZaFunkcTestA.ResetStep:= TRUE;
				SC_P4_ZdvizkaZaFunkcTestA.Step:= 100;
			END_IF

		//********************************************************Automatický režim****************************************************************************//

		100:
			SC_P4_ZdvizkaZaFunkcTestA.StepName:='100 - Automaticky Rezim - cakam na príchod paletky na zdvizku';
			SC_P4_ZdvizkaZaFunkcTestA.IdleTime.PT:= T#200ms;
			SC_P4_ZdvizkaZaFunkcTestA.AlarmTime.PT:= T#5s;

			SC_P4_ZdvizkaZaFunkcTestA.IdleTime.IN:= P4_ZdvizkaZaFunkcTestA.IN.PritomnostPaletky AND P4_ZdvizkaZaFunkcTestA.IN.PoziciaPaletky_OK AND P4_ZdvizkaZaFunkcTestA.IN.Zdvizka_StrednaPoloha;

			IF P4_ZdvizkaZaFunkcTestA.IN.PritomnostPaletky AND P4_ZdvizkaZaFunkcTestA.IN.PoziciaPaletky_OK THEN
				P4_FunkcnyTestA.STAV.PrebiehaVyvezeniePaletky:= FALSE;
				P4_ZdvizkaZaFunkcTestB.STAV.PrebiehaVyvezeniePaletky:= FALSE;
			END_IF

			IF P4_ZdvizkaZaFunkcTestA.KoniecCyklu AND NOT P4_FunkcnyTestA.Automat THEN
				SC_P4_ZdvizkaZaFunkcTestA.ResetStep:= TRUE;
				SC_P4_ZdvizkaZaFunkcTestA.Step:= 0;
			ELSIF SC_P4_ZdvizkaZaFunkcTestA.IdleTime.Q THEN
				SC_P4_ZdvizkaZaFunkcTestA.ResetStep:= TRUE;
				SC_P4_ZdvizkaZaFunkcTestA.Step:= 101;
			END_IF

		101:
			SC_P4_ZdvizkaZaFunkcTestA.StepName:='101 - Automaticky Rezim - cakam na vyvezenie na trat A';
			SC_P4_ZdvizkaZaFunkcTestA.IdleTime.PT:= T#200ms;
			SC_P4_ZdvizkaZaFunkcTestA.AlarmTime.PT:= T#5s;

			IF P4_ZdvizkaZaFunkcTestA.KoniecCyklu AND NOT P4_FunkcnyTestA.Automat AND NOT P4_ZdvizkaZaFunkcTestB.Automat THEN
				SC_P4_ZdvizkaZaFunkcTestA.ResetStep:= TRUE;
				SC_P4_ZdvizkaZaFunkcTestA.Step:= 0;
			ELSIF NOT P4_Etiketovacka.RFID_hlava.PritomnostPaletky AND SC_P4_Etiketovacka.Step = 100 AND NOT P4_ZdvizkaZaFunkcTestA.STAV.PrebiehaVyvezeniePaletky AND NOT P4_ZdvizkaZaFunkcTestB.STAV.PrebiehaVyvezeniePaletky THEN
				SC_P4_ZdvizkaZaFunkcTestA.ResetStep:= TRUE;
				SC_P4_ZdvizkaZaFunkcTestA.Step:= 110;
			END_IF

		//Vyvážanie na trať A//

		110:
			SC_P4_ZdvizkaZaFunkcTestA.StepName:='110 - Automaticky Rezim - presun zdvizky do spodnej polohy';
			SC_P4_ZdvizkaZaFunkcTestA.IdleTime.PT:= T#200ms;
			SC_P4_ZdvizkaZaFunkcTestA.AlarmTime.PT:= T#5s;

			IF NOT SC_P4_ZdvizkaZaFunkcTestA.Switch1 AND SC_OvlZdvizky.Step = 1 THEN
				Zdvizku_ZASUN:= TRUE;
				P4_ZdvizkaZaFunkcTestA.STAV.PrebiehaVyvezeniePaletky:= TRUE;
				SC_P4_ZdvizkaZaFunkcTestA.Switch1:= TRUE;
			END_IF

			IF P4_ZdvizkaZaFunkcTestA.IN.Zdvizka_SpodnaPoloha THEN
				SC_P4_ZdvizkaZaFunkcTestA.ResetStep:= TRUE;
				SC_P4_ZdvizkaZaFunkcTestA.Step:= 113;
			END_IF

		113:
			SC_P4_ZdvizkaZaFunkcTestA.StepName:='113 - Automaticky Rezim - cakam na ukoncenie vyvazania na Trat A';
			SC_P4_ZdvizkaZaFunkcTestA.IdleTime.PT:= T#500ms;
			SC_P4_ZdvizkaZaFunkcTestA.AlarmTime.PT:= T#5s;

			IF P4_Etiketovacka.RFID_hlava.PritomnostPaletky AND NOT SC_P4_ZdvizkaZaFunkcTestA.Switch1 AND SC_OvlZdvizky.Step = 1 THEN
				Zdvizku_VYSTRED:= TRUE;
				SC_P4_ZdvizkaZaFunkcTestA.Switch1:= TRUE;
			END_IF

			IF P4_ZdvizkaZaFunkcTestA.IN.Zdvizka_StrednaPoloha THEN
				SC_P4_ZdvizkaZaFunkcTestA.ResetStep:= TRUE;
				SC_P4_ZdvizkaZaFunkcTestA.Step:= 130;
			END_IF

			//Vysunutie tlmenia paletky//

		130:
			SC_P4_ZdvizkaZaFunkcTestA.StepName:='130 - Automaticky Rezim - vysunutie tlamena paletky';
			SC_P4_ZdvizkaZaFunkcTestA.IdleTime.PT:= T#1s;
			SC_P4_ZdvizkaZaFunkcTestA.AlarmTime.PT:= T#5s;

			SC_P4_ZdvizkaZaFunkcTestA.IdleTime.IN:= NOT P4_ZdvizkaZaFunkcTestA.IN.TlmicPaletky_ZASUNUTY;

			IF NOT SC_P4_ZdvizkaZaFunkcTestA.Switch1 THEN
				P4_ZdvizkaZaFunkcTestA.OUT.TlmicPaletky_ZASUN:= FALSE;
				P4_ZdvizkaZaFunkcTestA.OUT.TlmicPaletky_VYSUN:= TRUE;
				SC_P4_ZdvizkaZaFunkcTestA.Switch1:= TRUE;
			END_IF

			IF SC_P4_ZdvizkaZaFunkcTestA.IdleTime.Q THEN
				P4_ZdvizkaZaFunkcTestA.OUT.TlmicPaletky_ZASUN:= FALSE;
				P4_ZdvizkaZaFunkcTestA.OUT.TlmicPaletky_VYSUN:= FALSE;
				SC_P4_ZdvizkaZaFunkcTestA.ResetStep:= TRUE;
				SC_P4_ZdvizkaZaFunkcTestA.Step:= 100;
			END_IF

			//*******************************************************Manuálny režim*******************************************************************************//
		700:
			SC_P4_ZdvizkaZaFunkcTestA.StepName:='700 - Manualny Rezim';
			SC_P4_ZdvizkaZaFunkcTestA.IdleTime.PT:= T#8s;
			SC_P4_ZdvizkaZaFunkcTestA.AlarmTime.PT:= T#5s;

	END_CASE

END_PROGRAM

PROGRAM _EXIT
	(* Insert code here *)

END_PROGRAM
```

#### Variables.var - Local variables
```iecst
VAR
	SC_OvlZdvizky : SequenceControlTyp;
	Zdvizku_VYSUN : BOOL;
	Zdvizku_ZASUN : BOOL;
	Zdvizku_VYSTRED : BOOL := FALSE;
END_VAR
```

#### OvlZdvizky.st
```iecst
ACTION OvlZdvizky:

	//Volanie funkcie SequenceControl//
	SequenceControl(SC:= SC_OvlZdvizky);

	CASE SC_OvlZdvizky.Step OF

		0:
			SC_OvlZdvizky.StepName:= '0 - Nulovanie';
			Zdvizku_VYSUN:= FALSE;
			Zdvizku_ZASUN:= FALSE;
			Zdvizku_VYSTRED:= FALSE;

			IF SC_P4_ZdvizkaZaFunkcTestA.Step <> 0 THEN
				SC_OvlZdvizky.ResetStep:= TRUE;
				SC_OvlZdvizky.Step:= 1;
			END_IF

		1:
			SC_OvlZdvizky.StepName:= '1 - Rozhodnutie o cinnosti';
			IF Zdvizku_VYSUN THEN
				SC_OvlZdvizky.Step:= 10;
			ELSIF Zdvizku_ZASUN THEN
				SC_OvlZdvizky.Step:= 20;
			ELSIF Zdvizku_VYSTRED THEN
				SC_OvlZdvizky.Step:= 30;
			END_IF

		10:
			SC_OvlZdvizky.StepName:= '10 - Vysunutie zdvizky hore';
			SC_OvlZdvizky.IdleTime.PT:= T#3s;
			SC_OvlZdvizky.AlarmTime.PT:= T#6s;

			IF P4_ZdvizkaZaFunkcTestA.Automat THEN
				SC_OvlZdvizky.AlarmTime.IN:= TRUE;
			ELSE
				SC_OvlZdvizky.IdleTime.IN:= TRUE;
			END_IF

			IF NOT SC_OvlZdvizky.Switch1 THEN
				P4_ZdvizkaZaFunkcTestA.OUT.Zdvizku_ZASUN:= FALSE;
				P4_ZdvizkaZaFunkcTestA.OUT.Zdvizku_VYSUN:= TRUE;
				SC_OvlZdvizky.Switch1:= TRUE;
			END_IF

			IF P4_ZdvizkaZaFunkcTestA.IN.Zdvizka_HornaPoloha OR SC_OvlZdvizky.IdleTime.Q THEN
				SC_OvlZdvizky.ResetStep:= TRUE;
				SC_OvlZdvizky.Step:= 0;
			ELSIF SC_OvlZdvizky.AlarmTime.Q THEN
				P34_Alarmy[456]:= TRUE;
				P4_Pracovisko.STAV.Porucha_ST3:= TRUE;
			END_IF

		20:
			SC_OvlZdvizky.StepName:= '20 - Zasunutie zdvizky dole';
			SC_OvlZdvizky.IdleTime.PT:= T#3s;
			SC_OvlZdvizky.AlarmTime.PT:= T#6s;

			IF P4_ZdvizkaZaFunkcTestA.Automat THEN
				SC_OvlZdvizky.AlarmTime.IN:= TRUE;
			ELSE
				SC_OvlZdvizky.IdleTime.IN:= TRUE;
			END_IF

			IF NOT SC_OvlZdvizky.Switch1 THEN
				P4_ZdvizkaZaFunkcTestA.OUT.Zdvizku_VYSUN:= FALSE;
				P4_ZdvizkaZaFunkcTestA.OUT.Zdvizku_ZASUN:= TRUE;
				SC_OvlZdvizky.Switch1:= TRUE;
			END_IF

			IF P4_ZdvizkaZaFunkcTestA.IN.Zdvizka_SpodnaPoloha OR SC_OvlZdvizky.IdleTime.Q THEN
				SC_OvlZdvizky.ResetStep:= TRUE;
				SC_OvlZdvizky.Step:= 0;
			ELSIF SC_OvlZdvizky.AlarmTime.Q THEN
				P34_Alarmy[457]:= TRUE;
				P4_Pracovisko.STAV.Porucha_ST3:= TRUE;
			END_IF

		30:
			SC_OvlZdvizky.StepName:= '30 - Presun zdvizky do strednej polohy';
			SC_OvlZdvizky.IdleTime.PT:= T#3s;
			SC_OvlZdvizky.AlarmTime.PT:= T#6s;

			IF P4_ZdvizkaZaFunkcTestA.Automat THEN
				SC_OvlZdvizky.AlarmTime.IN:= TRUE;
			ELSE
				SC_OvlZdvizky.IdleTime.IN:= TRUE;
			END_IF

			IF NOT SC_OvlZdvizky.Switch1 THEN
				P4_ZdvizkaZaFunkcTestA.OUT.Zdvizku_VYSUN:= FALSE;
				P4_ZdvizkaZaFunkcTestA.OUT.Zdvizku_ZASUN:= FALSE;
				SC_OvlZdvizky.Switch1:= TRUE;
			END_IF

			IF P4_ZdvizkaZaFunkcTestA.IN.Zdvizka_StrednaPoloha OR SC_OvlZdvizky.IdleTime.Q THEN
				SC_OvlZdvizky.ResetStep:= TRUE;
				SC_OvlZdvizky.Step:= 0;
			ELSIF SC_OvlZdvizky.AlarmTime.Q THEN
				P34_Alarmy[458]:= TRUE;
				P4_Pracovisko.STAV.Porucha_ST3:= TRUE;
			END_IF

	END_CASE

END_ACTION
```

### Program Logical/Program/Pracovisko_4/P4_ZdvizkaZaFunkcTestB (IEC)

#### Main.st - Init, cyclic, exit code
```iecst
PROGRAM _INIT
	(* Insert code here *)

END_PROGRAM

PROGRAM _CYCLIC

	//Volanie funkcie SequenceControl//
	SequenceControl(SC:= SC_P4_ZdvizkaZaFunkcTestB);

	//Volanie podprogramov//
	OvlZdvizky;

	//Reset sekcie //
	IF P4_ZdvizkaZaFunkcTestB.Reset THEN
		SC_P4_ZdvizkaZaFunkcTestB.Step:= 0;
		P4_ZdvizkaZaFunkcTestB.Reset:= FALSE;
	ELSIF NOT Safety.STAV.Linka_ZonaCS_AKTIVNA THEN
		SC_P4_ZdvizkaZaFunkcTestB.Step:= 0;
	END_IF

	CASE SC_P4_ZdvizkaZaFunkcTestB.Step OF

		0:
			SC_P4_ZdvizkaZaFunkcTestB.StepName:='0 - Nulovanie';
			SC_OvlZdvizky.Step:= 0;
			P4_ZdvizkaZaFunkcTestB.Automat:= FALSE;
			P4_ZdvizkaZaFunkcTestB.KoniecCyklu:= FALSE;
			P4_ZdvizkaZaFunkcTestB.Manual:= FALSE;
			P4_ZdvizkaZaFunkcTestB.STAV.PoINIT:= FALSE;
			P4_ZdvizkaZaFunkcTestB.OUT.TlmicPaletky_VYSUN:= FALSE;

			P4_ZdvizkaZaFunkcTestB.STAV.PrebiehaVyvezeniePaletky:= FALSE;
			P4_FunkcnyTestB.STAV.PrebiehaVyvezeniePaletky:= FALSE;

			IF Safety.STAV.Linka_ZonaCS_AKTIVNA AND
				Safety.STAV.P4_ZonaBunky_AKTIVNA AND
				P4_Pracovisko.STAV.HardwareBunky_OK AND
				NOT P3_Pracovisko.STAV.Porucha_ST1 AND
				NOT P3_Pracovisko.STAV.Porucha_ST2 AND
				NOT P3_Pracovisko.STAV.Porucha_ST3 AND
				NOT P3_Pracovisko.STAV.Porucha_ST4 AND
				NOT P3_Pracovisko.STAV.Porucha_ST5 AND
				NOT P3_Pracovisko.STAV.Porucha_ST6 AND
				NOT P3_Pracovisko.STAV.Porucha_ST7 AND
				NOT P3_Pracovisko.STAV.Porucha_ST8 THEN
				SC_P4_ZdvizkaZaFunkcTestB.ResetStep:= TRUE;
				SC_P4_ZdvizkaZaFunkcTestB.Step:= 1;
			END_IF

		1:
			SC_P4_ZdvizkaZaFunkcTestB.StepName:='1 - Cakam na spustenie vyroby';
			P4_ZdvizkaZaFunkcTestB.KoniecCyklu:= FALSE;
			IF P4_ZdvizkaZaFunkcTestB.Automat THEN
				SC_P4_ZdvizkaZaFunkcTestB.Step:= 2;
			ELSIF P4_ZdvizkaZaFunkcTestB.Manual THEN
				SC_P4_ZdvizkaZaFunkcTestB.Step:= 700;
			END_IF

			//********************************************************Inicializácia****************************************************************************//

		2:
			SC_P4_ZdvizkaZaFunkcTestB.StepName:='2 - Inicializacia - cakam na spustenie inicializacie';
			SC_P4_ZdvizkaZaFunkcTestB.IdleTime.PT:= T#500ms;
			SC_P4_ZdvizkaZaFunkcTestB.AlarmTime.PT:= T#5s;

			IF P4_Dopravniky.STAV.PoINIT AND P4_ZdvizkaZaFunkcTestA.STAV.PoINIT THEN
				SC_P4_ZdvizkaZaFunkcTestB.ResetStep:= TRUE;
				SC_P4_ZdvizkaZaFunkcTestB.Step:= 5;
			END_IF

		5:
			SC_P4_ZdvizkaZaFunkcTestB.StepName:='5 - Inicializacia - kontrola pozicie zdvizky';
			SC_P4_ZdvizkaZaFunkcTestB.IdleTime.PT:= T#500ms;
			SC_P4_ZdvizkaZaFunkcTestB.AlarmTime.PT:= T#5s;

			IF P4_ZdvizkaZaFunkcTestB.IN.Zdvizka_StrednaPoloha AND P4_ZdvizkaZaFunkcTestB.IN.PritomnostPaletky THEN
				P4_ZdvizkaZaFunkcTestB.STAV.PoINIT:= TRUE;
				SC_P4_ZdvizkaZaFunkcTestB.ResetStep:= TRUE;
				SC_P4_ZdvizkaZaFunkcTestB.Step:= 100;
			ELSIF P4_ZdvizkaZaFunkcTestB.IN.Zdvizka_StrednaPoloha AND NOT P4_ZdvizkaZaFunkcTestB.IN.PritomnostPaletky THEN
				P4_ZdvizkaZaFunkcTestB.STAV.PoINIT:= TRUE;
				SC_P4_ZdvizkaZaFunkcTestB.ResetStep:= TRUE;
				SC_P4_ZdvizkaZaFunkcTestB.Step:= 100;
			ELSE
				SC_P4_ZdvizkaZaFunkcTestB.ResetStep:= TRUE;
				SC_P4_ZdvizkaZaFunkcTestB.Step:= 8;
			END_IF

		8:
			SC_P4_ZdvizkaZaFunkcTestB.StepName:='8 - Inicializacia - presun zdvizky do strednej polohy';
			SC_P4_ZdvizkaZaFunkcTestB.IdleTime.PT:= T#5s;
			SC_P4_ZdvizkaZaFunkcTestB.AlarmTime.PT:= T#5s;

			IF NOT SC_P4_ZdvizkaZaFunkcTestB.Switch1 AND SC_OvlZdvizky.Step = 1 THEN
				Zdvizku_VYSTRED:= TRUE;
				SC_P4_ZdvizkaZaFunkcTestB.Switch1:= TRUE;
			END_IF

			IF P4_ZdvizkaZaFunkcTestB.IN.Zdvizka_StrednaPoloha THEN
				SC_P4_ZdvizkaZaFunkcTestB.ResetStep:= TRUE;
				SC_P4_ZdvizkaZaFunkcTestB.Step:= 10;
			END_IF

		10:
			SC_P4_ZdvizkaZaFunkcTestB.StepName:='10 - Inicializacia - hladania paletky';
			SC_P4_ZdvizkaZaFunkcTestB.IdleTime.PT:= T#5s;
			SC_P4_ZdvizkaZaFunkcTestB.AlarmTime.PT:= T#5s;

			SC_P4_ZdvizkaZaFunkcTestB.IdleTime.IN:= TRUE;

			IF SC_P4_ZdvizkaZaFunkcTestB.IdleTime.Q THEN
				SC_P4_ZdvizkaZaFunkcTestB.ResetStep:= TRUE;
				SC_P4_ZdvizkaZaFunkcTestB.Step:= 5;
			END_IF

		//********************************************************Automatický režim****************************************************************************//

		100:
			SC_P4_ZdvizkaZaFunkcTestB.StepName:='100 - Automaticky Rezim - cakam na príchod paletky na zdvizku';
			SC_P4_ZdvizkaZaFunkcTestB.IdleTime.PT:= T#500ms;
			SC_P4_ZdvizkaZaFunkcTestB.AlarmTime.PT:= T#5s;

			SC_P4_ZdvizkaZaFunkcTestB.IdleTime.IN:= P4_ZdvizkaZaFunkcTestB.IN.PritomnostPaletky;

			IF P4_ZdvizkaZaFunkcTestB.IN.PritomnostPaletky THEN
				P4_FunkcnyTestB.STAV.PrebiehaVyvezeniePaletky:= FALSE;
			END_IF

			IF P4_ZdvizkaZaFunkcTestB.KoniecCyklu AND NOT P4_FunkcnyTestB.Automat THEN
				SC_P4_ZdvizkaZaFunkcTestB.ResetStep:= TRUE;
				SC_P4_ZdvizkaZaFunkcTestB.Step:= 0;
			ELSIF SC_P4_ZdvizkaZaFunkcTestB.IdleTime.Q THEN
				SC_P4_ZdvizkaZaFunkcTestB.ResetStep:= TRUE;
				SC_P4_ZdvizkaZaFunkcTestB.Step:= 101;
			END_IF

		101:
			SC_P4_ZdvizkaZaFunkcTestB.StepName:='101 - Automaticky Rezim - cakam na vyvezenie na trat A';
			SC_P4_ZdvizkaZaFunkcTestB.IdleTime.PT:= T#200ms;
			SC_P4_ZdvizkaZaFunkcTestB.AlarmTime.PT:= T#5s;

			IF P4_ZdvizkaZaFunkcTestB.KoniecCyklu AND NOT P4_FunkcnyTestB.Automat THEN
				SC_P4_ZdvizkaZaFunkcTestB.ResetStep:= TRUE;
				SC_P4_ZdvizkaZaFunkcTestB.Step:= 0;
			ELSIF NOT P4_ZdvizkaZaFunkcTestA.IN.PritomnostPaletky AND SC_P4_ZdvizkaZaFunkcTestA.Step = 100 AND NOT P4_FunkcnyTestA.STAV.PrebiehaVyvezeniePaletky AND SC_P4_FunkcnyTestA.Step < 560 THEN
				SC_P4_ZdvizkaZaFunkcTestB.ResetStep:= TRUE;
				SC_P4_ZdvizkaZaFunkcTestB.Step:= 110;
			END_IF

		//Vyvážanie na trať A//

		110:
			SC_P4_ZdvizkaZaFunkcTestB.StepName:='110 - Automaticky Rezim - presun zdviziek do hornej polohy';
			SC_P4_ZdvizkaZaFunkcTestB.IdleTime.PT:= T#200ms;
			SC_P4_ZdvizkaZaFunkcTestB.AlarmTime.PT:= T#5s;

			IF NOT SC_P4_ZdvizkaZaFunkcTestB.Switch1 AND SC_OvlZdvizky.Step = 1 THEN
				Zdvizku_VYSUN:= TRUE;
				P4_ZdvizkaZaFunkcTestA.OUT.Zdvizku_ZASUN:= FALSE;
				P4_ZdvizkaZaFunkcTestA.OUT.Zdvizku_VYSUN:= TRUE;
				P4_ZdvizkaZaFunkcTestA.OUT.TlmicPaletky_VYSUN:= FALSE;
				P4_ZdvizkaZaFunkcTestA.OUT.TlmicPaletky_ZASUN:= TRUE;
				P4_ZdvizkaZaFunkcTestB.STAV.PrebiehaVyvezeniePaletky:= TRUE;
				SC_P4_ZdvizkaZaFunkcTestB.Switch1:= TRUE;
			END_IF

			IF P4_ZdvizkaZaFunkcTestA.IN.Zdvizka_HornaPoloha AND P4_ZdvizkaZaFunkcTestB.IN.Zdvizka_HornaPoloha AND P4_ZdvizkaZaFunkcTestA.IN.TlmicPaletky_ZASUNUTY THEN
				SC_P4_ZdvizkaZaFunkcTestB.ResetStep:= TRUE;
				SC_P4_ZdvizkaZaFunkcTestB.Step:= 113;
			END_IF

		113:
			SC_P4_ZdvizkaZaFunkcTestB.StepName:='113 - Automaticky Rezim - cakam na ukoncenie vyvazania na Trat A';
			SC_P4_ZdvizkaZaFunkcTestB.IdleTime.PT:= T#500ms;
			SC_P4_ZdvizkaZaFunkcTestB.AlarmTime.PT:= T#5s;

			SC_P4_ZdvizkaZaFunkcTestB.IdleTime.IN:= P4_ZdvizkaZaFunkcTestA.IN.PritomnostPaletky;

			IF NOT SC_P4_ZdvizkaZaFunkcTestB.Switch1 THEN
				P4_Dopravniky.OUT.PriecnyDopravnik_VPRED:= TRUE;
				SC_P4_ZdvizkaZaFunkcTestB.Switch1:= TRUE;
			END_IF

			IF SC_P4_ZdvizkaZaFunkcTestB.IdleTime.Q THEN
				P4_Dopravniky.OUT.PriecnyDopravnik_VPRED:= FALSE;
				SC_P4_ZdvizkaZaFunkcTestB.ResetStep:= TRUE;
				SC_P4_ZdvizkaZaFunkcTestB.Step:= 115;
			END_IF

		115:
			SC_P4_ZdvizkaZaFunkcTestB.StepName:='123 - Automaticky Rezim - cakam na presun zdviziek do strednej polohy';
			SC_P4_ZdvizkaZaFunkcTestB.IdleTime.PT:= T#1s;
			SC_P4_ZdvizkaZaFunkcTestB.AlarmTime.PT:= T#5s;

			IF NOT SC_P4_ZdvizkaZaFunkcTestB.Switch1 AND SC_OvlZdvizky.Step = 1 THEN
				Zdvizku_VYSTRED:= TRUE;
				P4_ZdvizkaZaFunkcTestA.OUT.Zdvizku_ZASUN:= FALSE;
				P4_ZdvizkaZaFunkcTestA.OUT.Zdvizku_VYSUN:= FALSE;
				SC_P4_ZdvizkaZaFunkcTestB.Switch1:= TRUE;
			END_IF

			IF P4_ZdvizkaZaFunkcTestA.IN.Zdvizka_StrednaPoloha AND P4_ZdvizkaZaFunkcTestB.IN.Zdvizka_StrednaPoloha THEN
				P4_ZdvizkaZaFunkcTestB.STAV.PrebiehaVyvezeniePaletky:= FALSE;
				SC_P4_ZdvizkaZaFunkcTestB.ResetStep:= TRUE;
				SC_P4_ZdvizkaZaFunkcTestB.Step:= 130;
			END_IF

			//Vysunutie tlmenia paletky//

		130:
			SC_P4_ZdvizkaZaFunkcTestB.StepName:='130 - Automaticky Rezim - vysunutie tlamena paletky';
			SC_P4_ZdvizkaZaFunkcTestB.IdleTime.PT:= T#1s;
			SC_P4_ZdvizkaZaFunkcTestB.AlarmTime.PT:= T#5s;

			IF NOT SC_P4_ZdvizkaZaFunkcTestB.Switch1 THEN
				P4_ZdvizkaZaFunkcTestB.OUT.TlmicPaletky_VYSUN:= TRUE;
				SC_P4_ZdvizkaZaFunkcTestB.IdleTime.IN:= TRUE;
				SC_P4_ZdvizkaZaFunkcTestB.Switch1:= TRUE;
			END_IF

			IF SC_P4_ZdvizkaZaFunkcTestB.IdleTime.Q THEN
				P4_ZdvizkaZaFunkcTestB.OUT.TlmicPaletky_VYSUN:= FALSE;
				SC_P4_ZdvizkaZaFunkcTestB.ResetStep:= TRUE;
				SC_P4_ZdvizkaZaFunkcTestB.Step:= 100;
			END_IF

			//*******************************************************Manuálny režim*******************************************************************************//
		700:
			SC_P4_ZdvizkaZaFunkcTestB.StepName:='700 - Manualny Rezim';
			SC_P4_ZdvizkaZaFunkcTestB.IdleTime.PT:= T#8s;
			SC_P4_ZdvizkaZaFunkcTestB.AlarmTime.PT:= T#5s;

	END_CASE

END_PROGRAM

PROGRAM _EXIT
	(* Insert code here *)

END_PROGRAM
```

#### Variables.var - Local variables
```iecst
VAR
	SC_OvlZdvizky : SequenceControlTyp;
	Zdvizku_VYSUN : BOOL;
	Zdvizku_ZASUN : BOOL;
	Zdvizku_VYSTRED : BOOL := FALSE;
END_VAR
```

#### OvlZdvizky.st
```iecst
ACTION OvlZdvizky:

	//Volanie funkcie SequenceControl//
	SequenceControl(SC:= SC_OvlZdvizky);

	CASE SC_OvlZdvizky.Step OF

		0:
			SC_OvlZdvizky.StepName:= '0 - Nulovanie';
			Zdvizku_VYSUN:= FALSE;
			Zdvizku_ZASUN:= FALSE;
			Zdvizku_VYSTRED:= FALSE;

			IF SC_P4_ZdvizkaZaFunkcTestB.Step <> 0 THEN
				SC_OvlZdvizky.ResetStep:= TRUE;
				SC_OvlZdvizky.Step:= 1;
			END_IF

		1:
			SC_OvlZdvizky.StepName:= '1 - Rozhodnutie o cinnosti';
			IF Zdvizku_VYSUN THEN
				SC_OvlZdvizky.Step:= 10;
			ELSIF Zdvizku_VYSTRED THEN
				SC_OvlZdvizky.Step:= 30;
			END_IF

		10:
			SC_OvlZdvizky.StepName:= '10 - Vysunutie zdvizky hore';
			SC_OvlZdvizky.IdleTime.PT:= T#3s;
			SC_OvlZdvizky.AlarmTime.PT:= T#6s;

			IF P4_ZdvizkaZaFunkcTestB.Automat THEN
				SC_OvlZdvizky.AlarmTime.IN:= TRUE;
			ELSE
				SC_OvlZdvizky.IdleTime.IN:= TRUE;
			END_IF

			IF NOT SC_OvlZdvizky.Switch1 THEN
				P4_ZdvizkaZaFunkcTestB.OUT.Zdvizku_VYSUN:= TRUE;
				SC_OvlZdvizky.Switch1:= TRUE;
			END_IF

			IF P4_ZdvizkaZaFunkcTestB.IN.Zdvizka_HornaPoloha OR SC_OvlZdvizky.IdleTime.Q THEN
				SC_OvlZdvizky.ResetStep:= TRUE;
				SC_OvlZdvizky.Step:= 0;
			ELSIF SC_OvlZdvizky.AlarmTime.Q THEN
				P34_Alarmy[459]:= TRUE;
				P4_Pracovisko.STAV.Porucha_ST4:= TRUE;
			END_IF

		30:
			SC_OvlZdvizky.StepName:= '30 - Presun zdvizky do strednej polohy';
			SC_OvlZdvizky.IdleTime.PT:= T#3s;
			SC_OvlZdvizky.AlarmTime.PT:= T#6s;

			IF P4_ZdvizkaZaFunkcTestB.Automat THEN
				SC_OvlZdvizky.AlarmTime.IN:= TRUE;
			ELSE
				SC_OvlZdvizky.IdleTime.IN:= TRUE;
			END_IF

			IF NOT SC_OvlZdvizky.Switch1 THEN
				P4_ZdvizkaZaFunkcTestB.OUT.Zdvizku_VYSUN:= FALSE;
				SC_OvlZdvizky.Switch1:= TRUE;
			END_IF

			IF P4_ZdvizkaZaFunkcTestB.IN.Zdvizka_StrednaPoloha OR SC_OvlZdvizky.IdleTime.Q THEN
				SC_OvlZdvizky.ResetStep:= TRUE;
				SC_OvlZdvizky.Step:= 0;
			ELSIF SC_OvlZdvizky.AlarmTime.Q THEN
				P34_Alarmy[461]:= TRUE;
				P4_Pracovisko.STAV.Porucha_ST4:= TRUE;
			END_IF

	END_CASE

END_ACTION
```

### Program Logical/Program/Pracovisko_4/P4_StoperEtiketovania (IEC)
